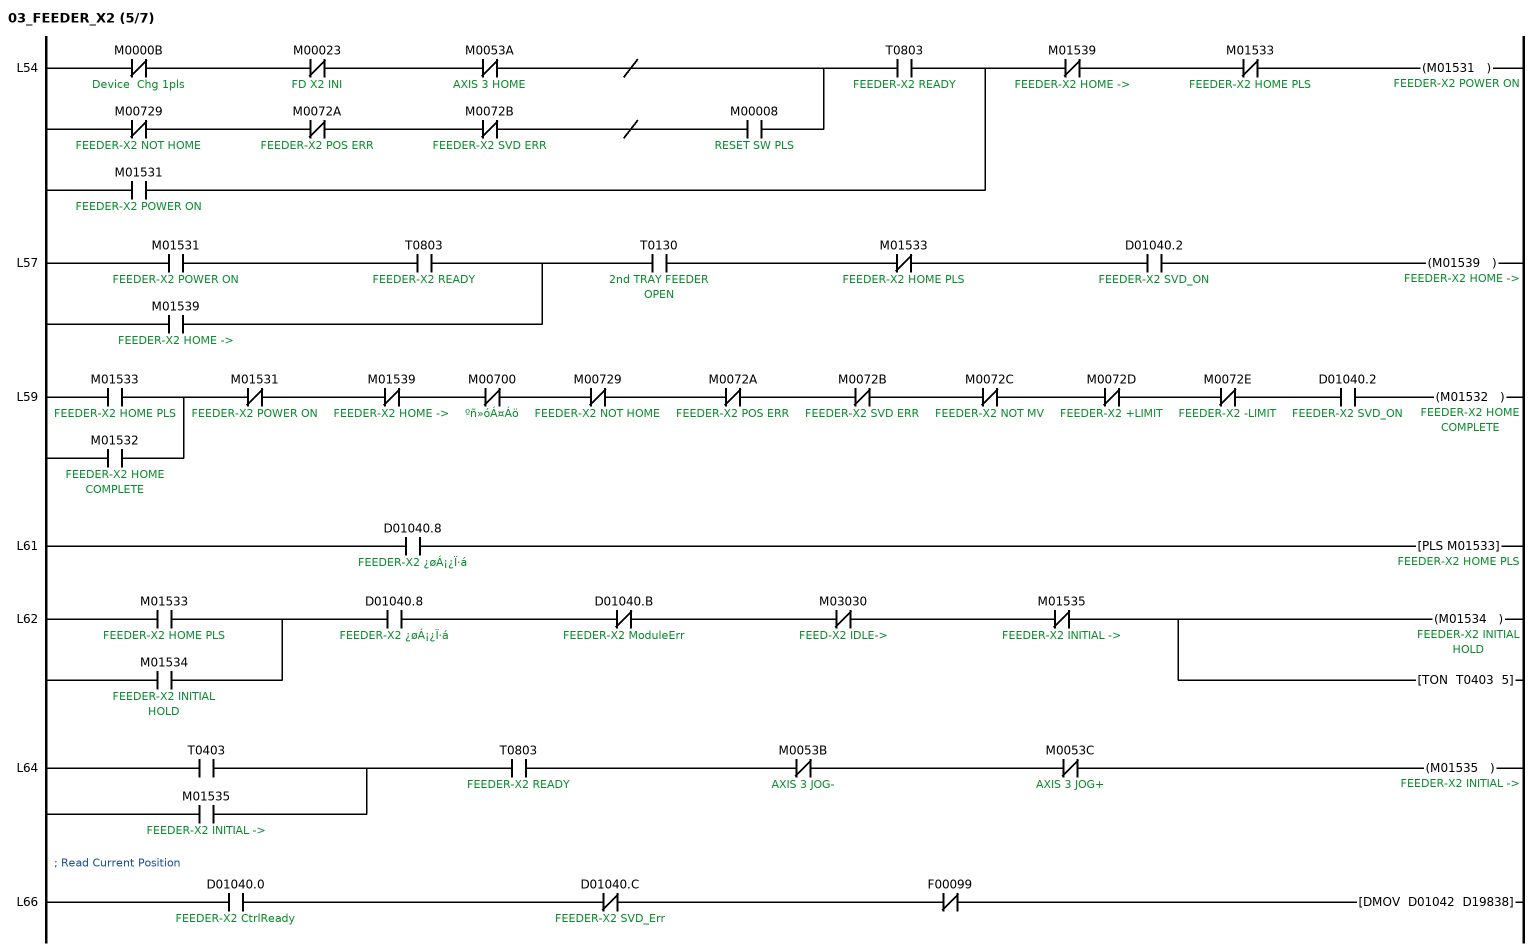
[picture p24: 03_FEEDER_X2 rungs L54-L66]
; L54
LOAD NOT  M0000B	// Device  Chg 1pls
AND NOT   M00023	// FD X2 INI
AND NOT   M0053A	// AXIS 3 HOME
NOT
LOAD NOT  M00729	// FEEDER-X2 NOT HOME
AND NOT   M0072A	// FEEDER-X2 POS ERR
AND NOT   M0072B	// FEEDER-X2 SVD ERR
NOT
AND       M00008	// RESET SW PLS
OR LOAD
AND       T0803	// FEEDER-X2 READY
OR        M01531	// FEEDER-X2 POWER ON
AND NOT   M01539	// FEEDER-X2 HOME ->
AND NOT   M01533	// FEEDER-X2 HOME PLS
OUT       M01531	// FEEDER-X2 POWER ON
; L57
LOAD      M01531	// FEEDER-X2 POWER ON
AND       T0803	// FEEDER-X2 READY
OR        M01539	// FEEDER-X2 HOME ->
AND       T0130	// 2nd TRAY FEEDER OPEN
AND NOT   M01533	// FEEDER-X2 HOME PLS
AND       D01040.2	// FEEDER-X2 SVD_ON
OUT       M01539	// FEEDER-X2 HOME ->
; L59
LOAD      M01533	// FEEDER-X2 HOME PLS
OR        M01532	// FEEDER-X2 HOME COMPLETE
AND NOT   M01531	// FEEDER-X2 POWER ON
AND NOT   M01539	// FEEDER-X2 HOME ->
AND NOT   M00700	// ºñ»óÁ¤Áö
AND NOT   M00729	// FEEDER-X2 NOT HOME
AND NOT   M0072A	// FEEDER-X2 POS ERR
AND NOT   M0072B	// FEEDER-X2 SVD ERR
AND NOT   M0072C	// FEEDER-X2 NOT MV
AND NOT   M0072D	// FEEDER-X2 +LIMIT
AND NOT   M0072E	// FEEDER-X2 -LIMIT
AND       D01040.2	// FEEDER-X2 SVD_ON
OUT       M01532	// FEEDER-X2 HOME COMPLETE
; L61
LOAD      D01040.8	// FEEDER-X2 ¿øÁ¡¿Ï·á
OUTP      M01533	// FEEDER-X2 HOME PLS
; L62
LOAD      M01533	// FEEDER-X2 HOME PLS
OR        M01534	// FEEDER-X2 INITIAL HOLD
AND       D01040.8	// FEEDER-X2 ¿øÁ¡¿Ï·á
AND NOT   D01040.B	// FEEDER-X2 ModuleErr
AND NOT   M03030	// FEED-X2 IDLE->
AND NOT   M01535	// FEEDER-X2 INITIAL ->
OUT       M01534	// FEEDER-X2 INITIAL HOLD
TON       T0403 5
; L64
LOAD      T0403
OR        M01535	// FEEDER-X2 INITIAL ->
AND       T0803	// FEEDER-X2 READY
AND NOT   M0053B	// AXIS 3 JOG-
AND NOT   M0053C	// AXIS 3 JOG+
OUT       M01535	// FEEDER-X2 INITIAL ->
; L66
LOAD      D01040.0	// FEEDER-X2 CtrlReady
AND NOT   D01040.C	// FEEDER-X2 SVD_Err
AND NOT   F00099
DMOV      D01042 D19838
// output comment: Read Current Position

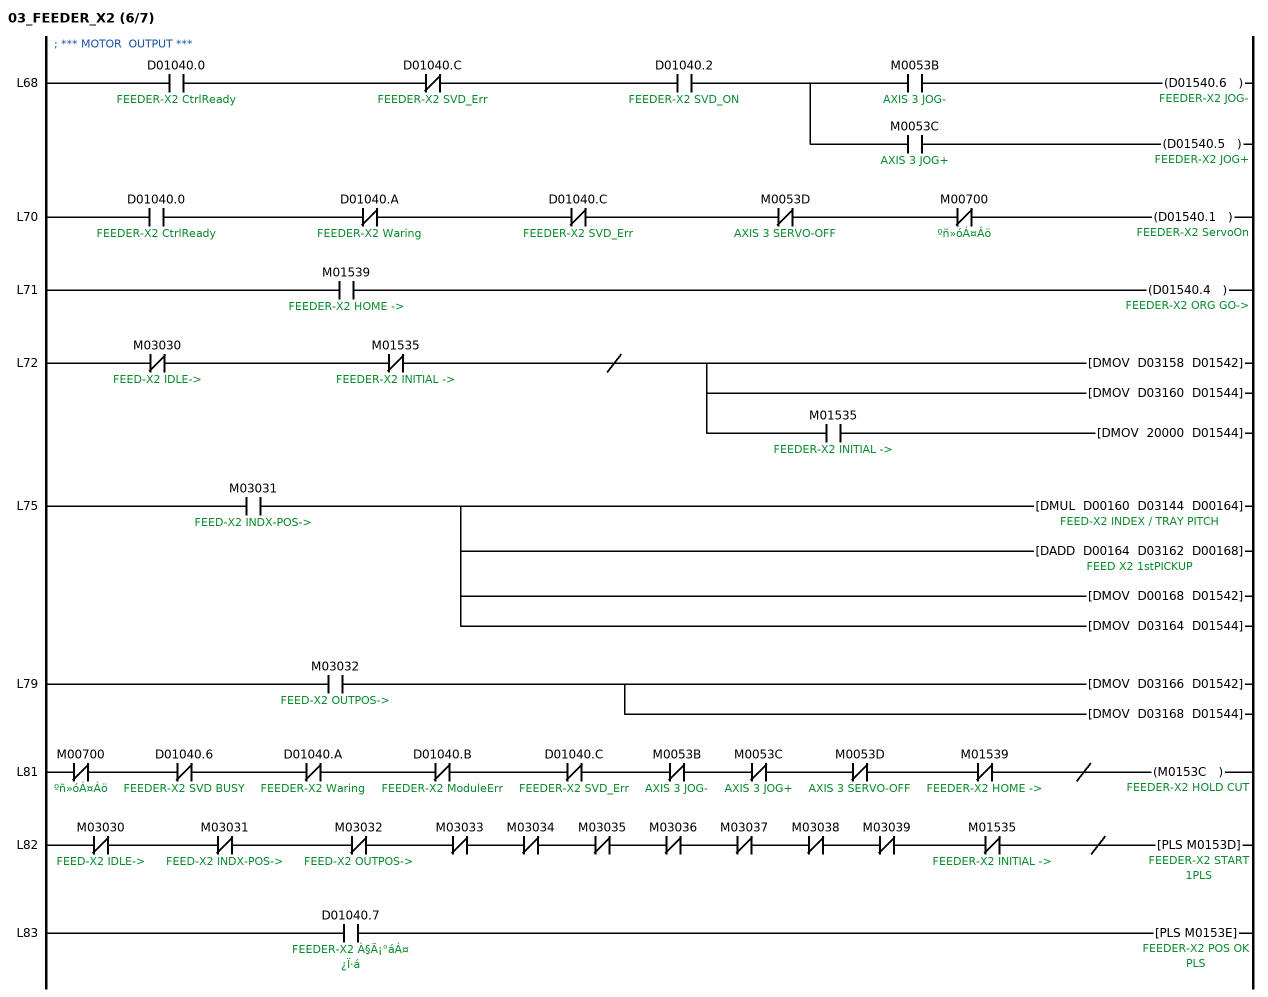
// *** MOTOR  OUTPUT ***
; L68
LOAD      D01040.0	// FEEDER-X2 CtrlReady
AND NOT   D01040.C	// FEEDER-X2 SVD_Err
AND       D01040.2	// FEEDER-X2 SVD_ON
MPUSH
AND       M0053B	// AXIS 3 JOG-
OUT       D01540.6	// FEEDER-X2 JOG-
MPOP
AND       M0053C	// AXIS 3 JOG+
OUT       D01540.5	// FEEDER-X2 JOG+
; L70
LOAD      D01040.0	// FEEDER-X2 CtrlReady
AND NOT   D01040.A	// FEEDER-X2 Waring
AND NOT   D01040.C	// FEEDER-X2 SVD_Err
AND NOT   M0053D	// AXIS 3 SERVO-OFF
AND NOT   M00700	// ºñ»óÁ¤Áö
OUT       D01540.1	// FEEDER-X2 ServoOn
; L71
LOAD      M01539	// FEEDER-X2 HOME ->
OUT       D01540.4	// FEEDER-X2 ORG GO->
; L72
LOAD NOT  M03030	// FEED-X2 IDLE->
AND NOT   M01535	// FEEDER-X2 INITIAL ->
NOT
DMOV      D03158 D01542
DMOV      D03160 D01544
AND       M01535	// FEEDER-X2 INITIAL ->
DMOV      20000 D01544
; L75
LOAD      M03031	// FEED-X2 INDX-POS->
DMUL      D00160 D03144 D00164	// FEED-X2 INDEX / TRAY PITCH
DADD      D00164 D03162 D00168	// FEED X2 1stPICKUP
DMOV      D00168 D01542
DMOV      D03164 D01544
; L79
LOAD      M03032	// FEED-X2 OUTPOS->
DMOV      D03166 D01542
DMOV      D03168 D01544
; L81
LOAD NOT  M00700	// ºñ»óÁ¤Áö
AND NOT   D01040.6	// FEEDER-X2 SVD BUSY
AND NOT   D01040.A	// FEEDER-X2 Waring
AND NOT   D01040.B	// FEEDER-X2 ModuleErr
AND NOT   D01040.C	// FEEDER-X2 SVD_Err
AND NOT   M0053B	// AXIS 3 JOG-
AND NOT   M0053C	// AXIS 3 JOG+
AND NOT   M0053D	// AXIS 3 SERVO-OFF
AND NOT   M01539	// FEEDER-X2 HOME ->
NOT
OUT       M0153C	// FEEDER-X2 HOLD CUT
; L82
LOAD NOT  M03030	// FEED-X2 IDLE->
AND NOT   M03031	// FEED-X2 INDX-POS->
AND NOT   M03032	// FEED-X2 OUTPOS->
AND NOT   M03033
AND NOT   M03034
AND NOT   M03035
AND NOT   M03036
AND NOT   M03037
AND NOT   M03038
AND NOT   M03039
AND NOT   M01535	// FEEDER-X2 INITIAL ->
NOT
OUTP      M0153D	// FEEDER-X2 START 1PLS
; L83
LOAD      D01040.7	// FEEDER-X2 À§Ä¡°áÁ¤ ¿Ï·á
OUTP      M0153E	// FEEDER-X2 POS OK PLS

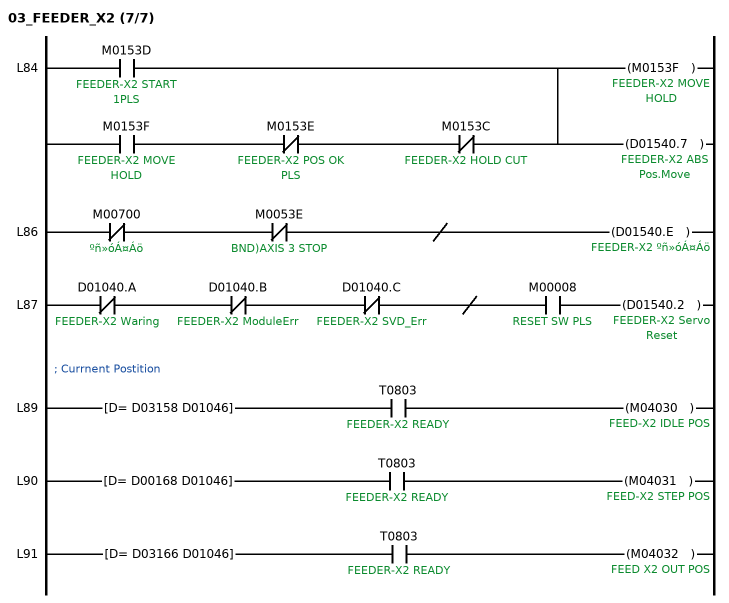
; L84
LOAD      M0153D	// FEEDER-X2 START 1PLS
LOAD      M0153F	// FEEDER-X2 MOVE HOLD
AND NOT   M0153E	// FEEDER-X2 POS OK PLS
AND NOT   M0153C	// FEEDER-X2 HOLD CUT
OR LOAD
OUT       M0153F	// FEEDER-X2 MOVE HOLD
OUT       D01540.7	// FEEDER-X2 ABS Pos.Move
; L86
LOAD NOT  M00700	// ºñ»óÁ¤Áö
AND NOT   M0053E	// BND)AXIS 3 STOP
NOT
OUT       D01540.E	// FEEDER-X2 ºñ»óÁ¤Áö
; L87
LOAD NOT  D01040.A	// FEEDER-X2 Waring
AND NOT   D01040.B	// FEEDER-X2 ModuleErr
AND NOT   D01040.C	// FEEDER-X2 SVD_Err
NOT
AND       M00008	// RESET SW PLS
OUT       D01540.2	// FEEDER-X2 Servo Reset
// Currnent Postition
; L89
LOADD=    D03158 D01046
AND       T0803	// FEEDER-X2 READY
OUT       M04030	// FEED-X2 IDLE POS
; L90
LOADD=    D00168 D01046
AND       T0803	// FEEDER-X2 READY
OUT       M04031	// FEED-X2 STEP POS
; L91
LOADD=    D03166 D01046
AND       T0803	// FEEDER-X2 READY
OUT       M04032	// FEED X2 OUT POS

PROGRAM 04_PICKER_Y (task: ½ºÄµ ÇÁ·Î±×·¥)

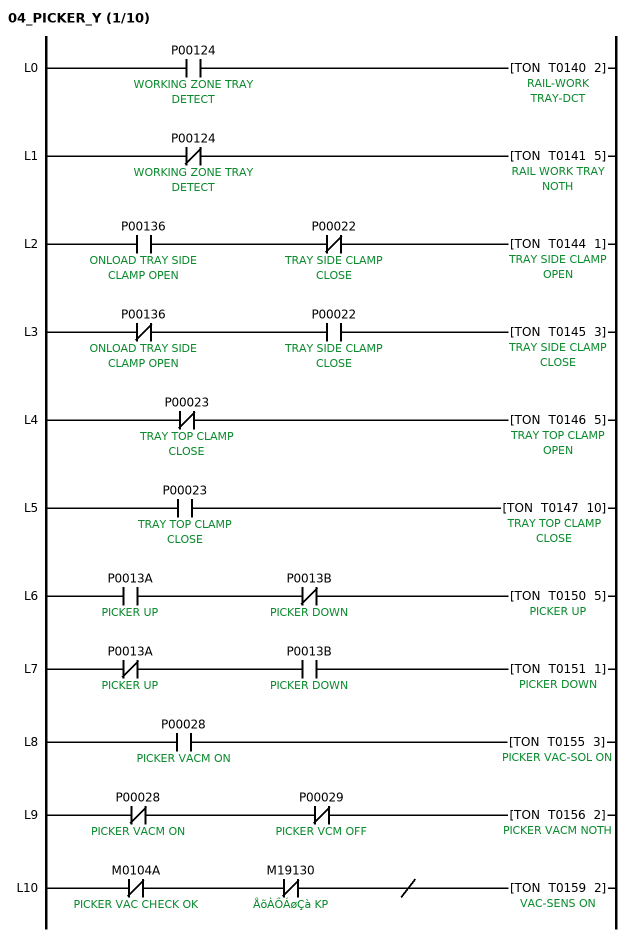
; L0
LOAD      P00124	// WORKING ZONE TRAY DETECT
TON       T0140 2	// RAIL-WORK TRAY-DCT
; L1
LOAD NOT  P00124	// WORKING ZONE TRAY DETECT
TON       T0141 5	// RAIL WORK TRAY NOTH
; L2
LOAD      P00136	// ONLOAD TRAY SIDE CLAMP OPEN
AND NOT   P00022	// TRAY SIDE CLAMP CLOSE
TON       T0144 1	// TRAY SIDE CLAMP OPEN
; L3
LOAD NOT  P00136	// ONLOAD TRAY SIDE CLAMP OPEN
AND       P00022	// TRAY SIDE CLAMP CLOSE
TON       T0145 3	// TRAY SIDE CLAMP CLOSE
; L4
LOAD NOT  P00023	// TRAY TOP CLAMP CLOSE
TON       T0146 5	// TRAY TOP CLAMP OPEN
; L5
LOAD      P00023	// TRAY TOP CLAMP CLOSE
TON       T0147 10	// TRAY TOP CLAMP CLOSE
; L6
LOAD      P0013A	// PICKER UP
AND NOT   P0013B	// PICKER DOWN
TON       T0150 5	// PICKER UP
; L7
LOAD NOT  P0013A	// PICKER UP
AND       P0013B	// PICKER DOWN
TON       T0151 1	// PICKER DOWN
; L8
LOAD      P00028	// PICKER VACM ON
TON       T0155 3	// PICKER VAC-SOL ON
; L9
LOAD NOT  P00028	// PICKER VACM ON
AND NOT   P00029	// PICKER VCM OFF
TON       T0156 2	// PICKER VACM NOTH
; L10
LOAD NOT  M0104A	// PICKER VAC CHECK OK
AND NOT   M19130	// ÅõÀÔÁøÇà KP
NOT
TON       T0159 2	// VAC-SENS ON

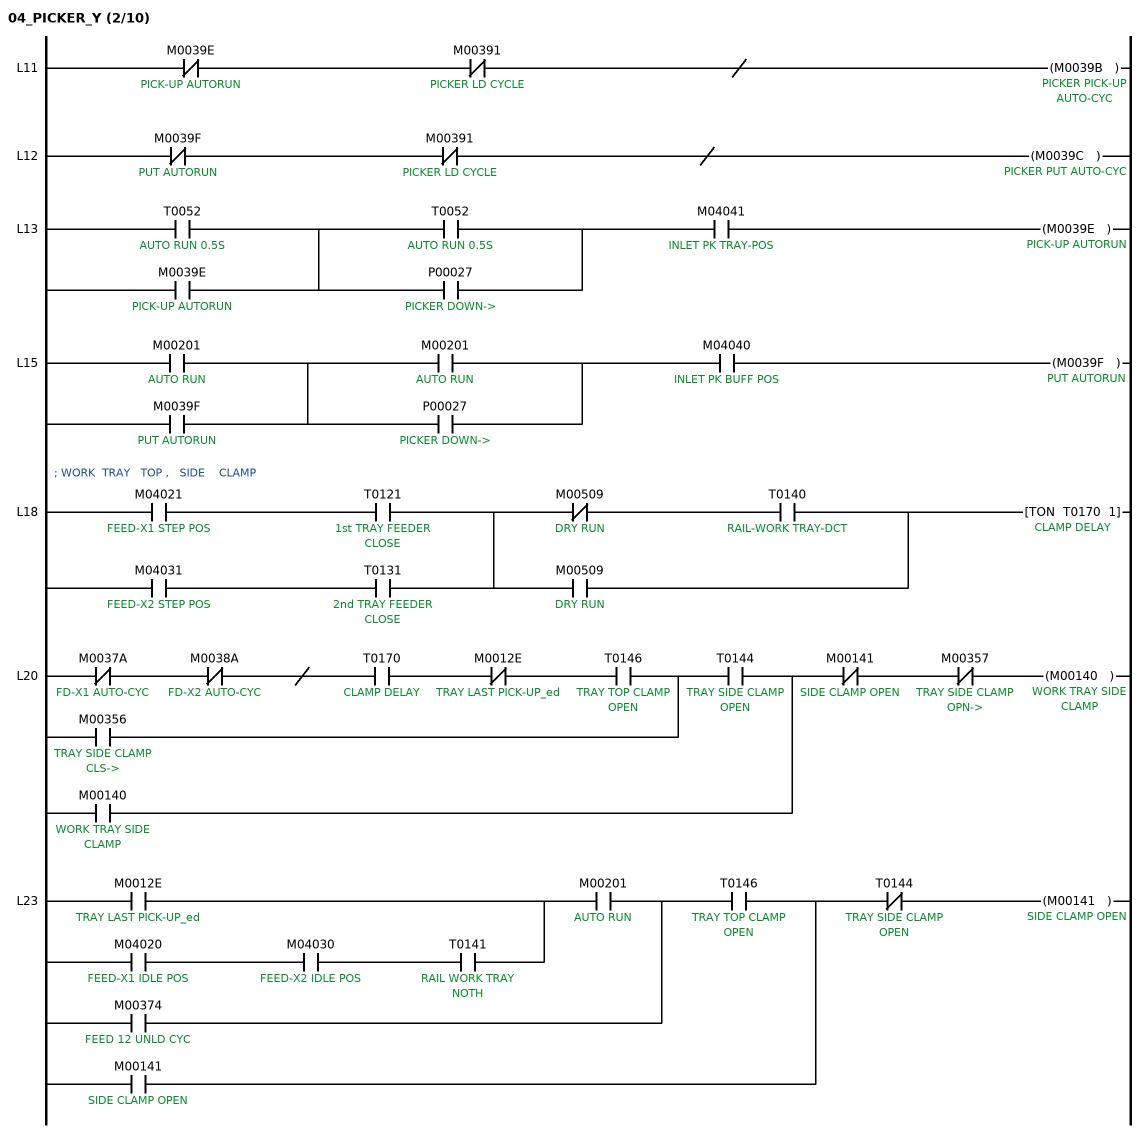
; L11
LOAD NOT  M0039E	// PICK-UP AUTORUN
AND NOT   M00391	// PICKER LD CYCLE
NOT
OUT       M0039B	// PICKER PICK-UP AUTO-CYC
; L12
LOAD NOT  M0039F	// PUT AUTORUN
AND NOT   M00391	// PICKER LD CYCLE
NOT
OUT       M0039C	// PICKER PUT AUTO-CYC
; L13
LOAD      T0052	// AUTO RUN 0.5S
OR        M0039E	// PICK-UP AUTORUN
LOAD      T0052	// AUTO RUN 0.5S
OR        P00027	// PICKER DOWN->
AND LOAD
AND       M04041	// INLET PK TRAY-POS
OUT       M0039E	// PICK-UP AUTORUN
; L15
LOAD      M00201	// AUTO RUN
OR        M0039F	// PUT AUTORUN
LOAD      M00201	// AUTO RUN
OR        P00027	// PICKER DOWN->
AND LOAD
AND       M04040	// INLET PK BUFF POS
OUT       M0039F	// PUT AUTORUN
// WORK  TRAY   TOP ,   SIDE    CLAMP
; L18
LOAD      M04021	// FEED-X1 STEP POS
AND       T0121	// 1st TRAY FEEDER CLOSE
LOAD      M04031	// FEED-X2 STEP POS
AND       T0131	// 2nd TRAY FEEDER CLOSE
OR LOAD
LOAD NOT  M00509	// DRY RUN
AND       T0140	// RAIL-WORK TRAY-DCT
OR        M00509	// DRY RUN
AND LOAD
TON       T0170 1	// CLAMP DELAY
; L20
LOAD NOT  M0037A	// FD-X1 AUTO-CYC
AND NOT   M0038A	// FD-X2 AUTO-CYC
NOT
AND       T0170	// CLAMP DELAY
AND NOT   M0012E	// TRAY LAST PICK-UP_ed
AND       T0146	// TRAY TOP CLAMP OPEN
OR        M00356	// TRAY SIDE CLAMP CLS->
AND       T0144	// TRAY SIDE CLAMP OPEN
OR        M00140	// WORK TRAY SIDE CLAMP
AND NOT   M00141	// SIDE CLAMP OPEN
AND NOT   M00357	// TRAY SIDE CLAMP OPN->
OUT       M00140	// WORK TRAY SIDE CLAMP
; L23
LOAD      M0012E	// TRAY LAST PICK-UP_ed
LOAD      M04020	// FEED-X1 IDLE POS
AND       M04030	// FEED-X2 IDLE POS
AND       T0141	// RAIL WORK TRAY NOTH
OR LOAD
AND       M00201	// AUTO RUN
OR        M00374	// FEED 12 UNLD CYC
AND       T0146	// TRAY TOP CLAMP OPEN
OR        M00141	// SIDE CLAMP OPEN
AND NOT   T0144	// TRAY SIDE CLAMP OPEN
OUT       M00141	// SIDE CLAMP OPEN

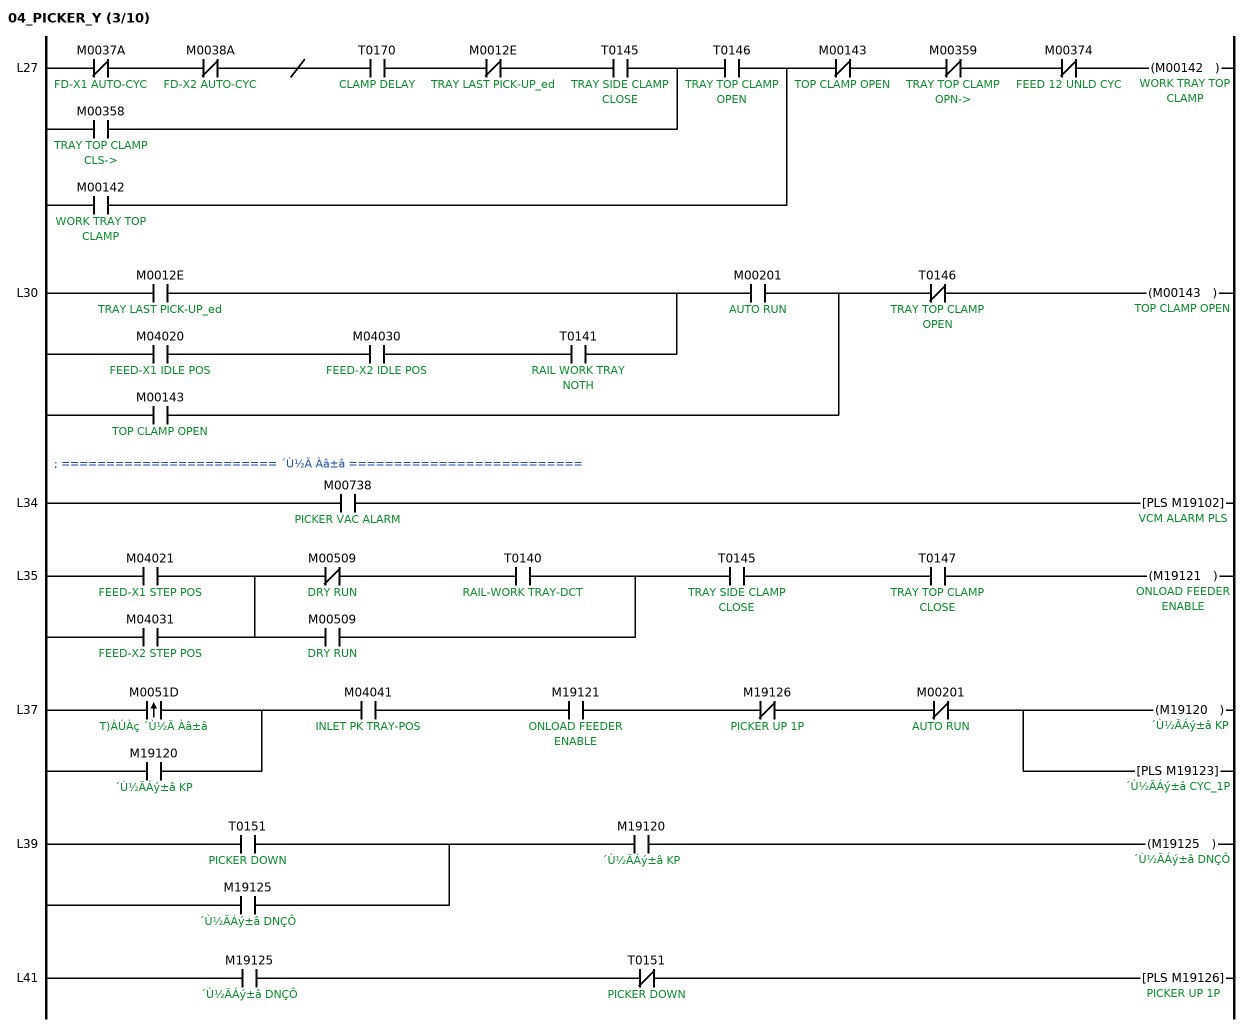
; L27
LOAD NOT  M0037A	// FD-X1 AUTO-CYC
AND NOT   M0038A	// FD-X2 AUTO-CYC
NOT
AND       T0170	// CLAMP DELAY
AND NOT   M0012E	// TRAY LAST PICK-UP_ed
AND       T0145	// TRAY SIDE CLAMP CLOSE
OR        M00358	// TRAY TOP CLAMP CLS->
AND       T0146	// TRAY TOP CLAMP OPEN
OR        M00142	// WORK TRAY TOP CLAMP
AND NOT   M00143	// TOP CLAMP OPEN
AND NOT   M00359	// TRAY TOP CLAMP OPN->
AND NOT   M00374	// FEED 12 UNLD CYC
OUT       M00142	// WORK TRAY TOP CLAMP
; L30
LOAD      M0012E	// TRAY LAST PICK-UP_ed
LOAD      M04020	// FEED-X1 IDLE POS
AND       M04030	// FEED-X2 IDLE POS
AND       T0141	// RAIL WORK TRAY NOTH
OR LOAD
AND       M00201	// AUTO RUN
OR        M00143	// TOP CLAMP OPEN
AND NOT   T0146	// TRAY TOP CLAMP OPEN
OUT       M00143	// TOP CLAMP OPEN
// ======================== ´Ù½Ã Àâ±â ==========================
; L34
LOAD      M00738	// PICKER VAC ALARM
OUTP      M19102	// VCM ALARM PLS
; L35
LOAD      M04021	// FEED-X1 STEP POS
OR        M04031	// FEED-X2 STEP POS
LOAD NOT  M00509	// DRY RUN
AND       T0140	// RAIL-WORK TRAY-DCT
OR        M00509	// DRY RUN
AND LOAD
AND       T0145	// TRAY SIDE CLAMP CLOSE
AND       T0147	// TRAY TOP CLAMP CLOSE
OUT       M19121	// ONLOAD FEEDER ENABLE
; L37
LOADP     M0051D	// T)ÀÚÀç ´Ù½Ã Àâ±â
OR        M19120	// ´Ù½ÃÁý±â KP
AND       M04041	// INLET PK TRAY-POS
AND       M19121	// ONLOAD FEEDER ENABLE
AND NOT   M19126	// PICKER UP 1P
AND NOT   M00201	// AUTO RUN
OUT       M19120	// ´Ù½ÃÁý±â KP
OUTP      M19123	// ´Ù½ÃÁý±â CYC_1P
; L39
LOAD      T0151	// PICKER DOWN
OR        M19125	// ´Ù½ÃÁý±â DNÇÔ
AND       M19120	// ´Ù½ÃÁý±â KP
OUT       M19125	// ´Ù½ÃÁý±â DNÇÔ
; L41
LOAD      M19125	// ´Ù½ÃÁý±â DNÇÔ
AND NOT   T0151	// PICKER DOWN
OUTP      M19126	// PICKER UP 1P

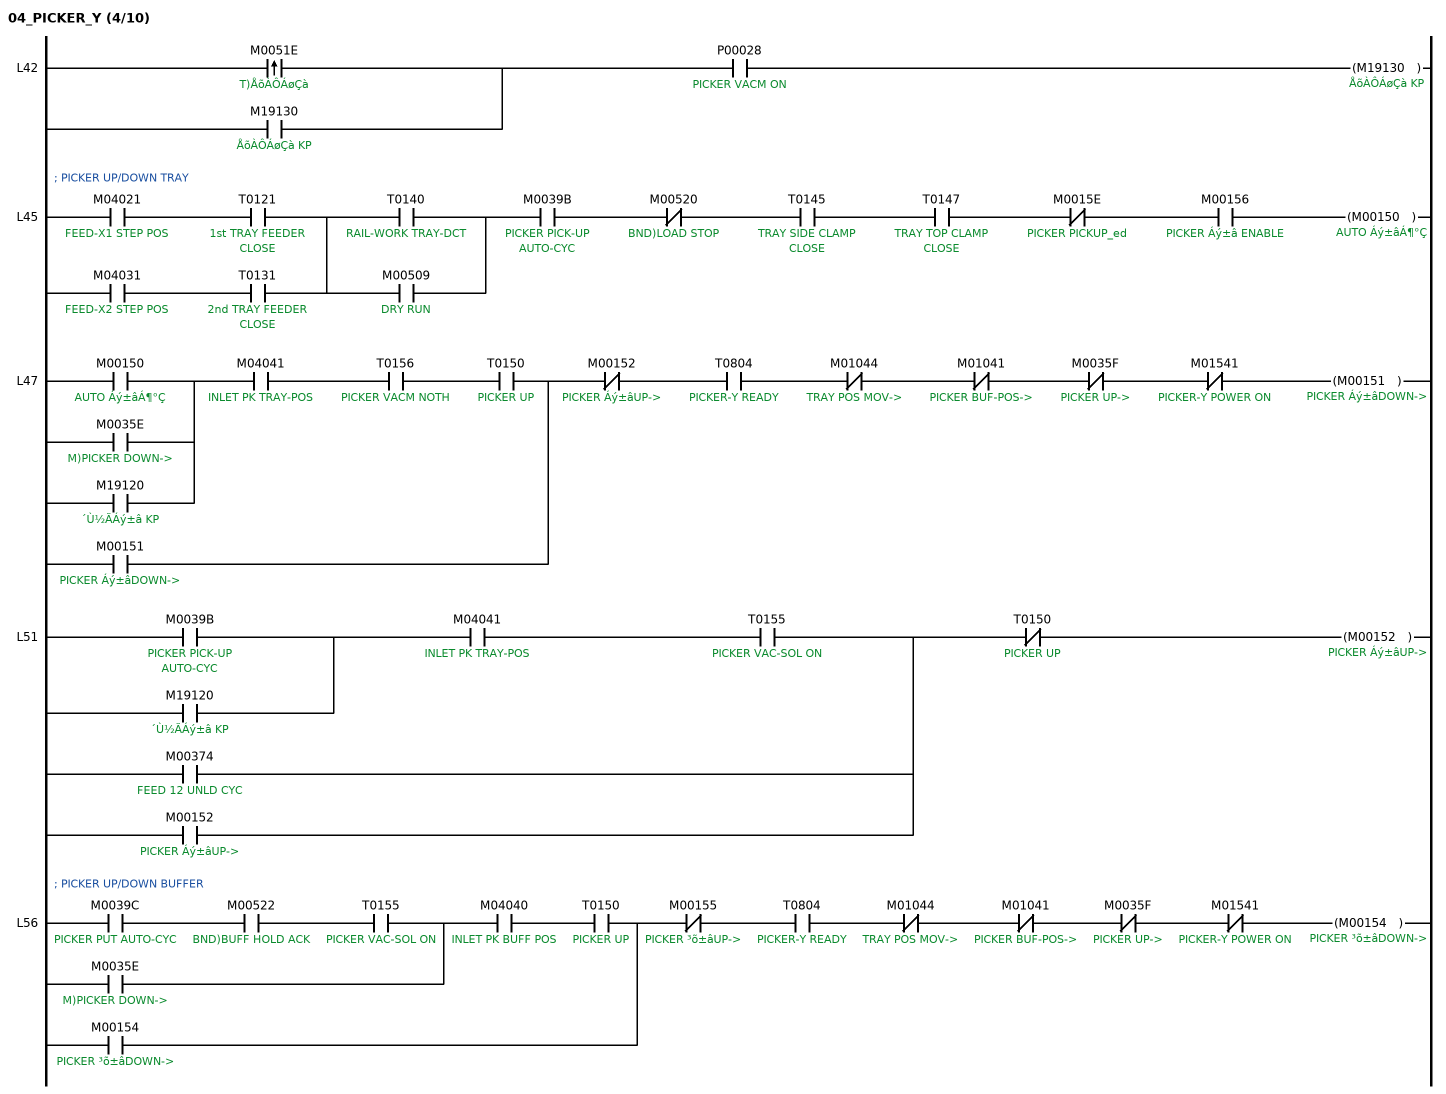
; L42
LOADP     M0051E	// T)ÅõÀÔÁøÇà
OR        M19130	// ÅõÀÔÁøÇà KP
AND       P00028	// PICKER VACM ON
OUT       M19130	// ÅõÀÔÁøÇà KP
// PICKER UP/DOWN TRAY
; L45
LOAD      M04021	// FEED-X1 STEP POS
AND       T0121	// 1st TRAY FEEDER CLOSE
LOAD      M04031	// FEED-X2 STEP POS
AND       T0131	// 2nd TRAY FEEDER CLOSE
OR LOAD
LOAD      T0140	// RAIL-WORK TRAY-DCT
OR        M00509	// DRY RUN
AND LOAD
AND       M0039B	// PICKER PICK-UP AUTO-CYC
AND NOT   M00520	// BND)LOAD STOP
AND       T0145	// TRAY SIDE CLAMP CLOSE
AND       T0147	// TRAY TOP CLAMP CLOSE
AND NOT   M0015E	// PICKER PICKUP_ed
AND       M00156	// PICKER Áý±â ENABLE
OUT       M00150	// AUTO Áý±âÁ¶°Ç
; L47
LOAD      M00150	// AUTO Áý±âÁ¶°Ç
OR        M0035E	// M)PICKER DOWN->
OR        M19120	// ´Ù½ÃÁý±â KP
AND       M04041	// INLET PK TRAY-POS
AND       T0156	// PICKER VACM NOTH
AND       T0150	// PICKER UP
OR        M00151	// PICKER Áý±âDOWN->
AND NOT   M00152	// PICKER Áý±âUP->
AND       T0804	// PICKER-Y READY
AND NOT   M01044	// TRAY POS MOV->
AND NOT   M01041	// PICKER BUF-POS->
AND NOT   M0035F	// PICKER UP->
AND NOT   M01541	// PICKER-Y POWER ON
OUT       M00151	// PICKER Áý±âDOWN->
; L51
LOAD      M0039B	// PICKER PICK-UP AUTO-CYC
OR        M19120	// ´Ù½ÃÁý±â KP
AND       M04041	// INLET PK TRAY-POS
AND       T0155	// PICKER VAC-SOL ON
OR        M00374	// FEED 12 UNLD CYC
OR        M00152	// PICKER Áý±âUP->
AND NOT   T0150	// PICKER UP
OUT       M00152	// PICKER Áý±âUP->
// PICKER UP/DOWN BUFFER
; L56
LOAD      M0039C	// PICKER PUT AUTO-CYC
AND       M00522	// BND)BUFF HOLD ACK
AND       T0155	// PICKER VAC-SOL ON
OR        M0035E	// M)PICKER DOWN->
AND       M04040	// INLET PK BUFF POS
AND       T0150	// PICKER UP
OR        M00154	// PICKER ³õ±âDOWN->
AND NOT   M00155	// PICKER ³õ±âUP->
AND       T0804	// PICKER-Y READY
AND NOT   M01044	// TRAY POS MOV->
AND NOT   M01041	// PICKER BUF-POS->
AND NOT   M0035F	// PICKER UP->
AND NOT   M01541	// PICKER-Y POWER ON
OUT       M00154	// PICKER ³õ±âDOWN->

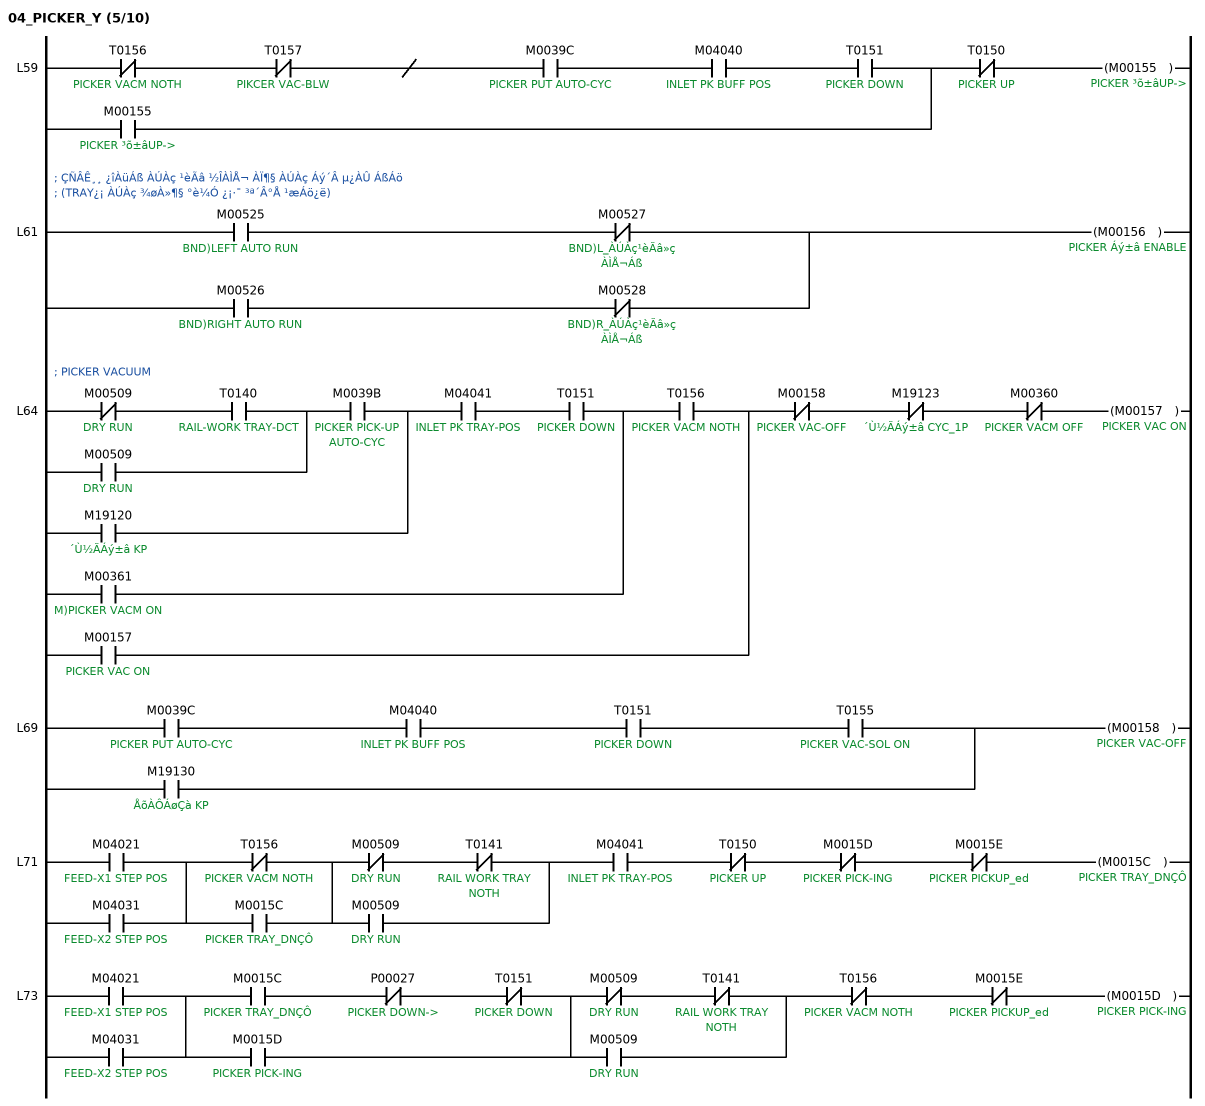
; L59
LOAD NOT  T0156	// PICKER VACM NOTH
AND NOT   T0157	// PIKCER VAC-BLW
NOT
AND       M0039C	// PICKER PUT AUTO-CYC
AND       M04040	// INLET PK BUFF POS
AND       T0151	// PICKER DOWN
OR        M00155	// PICKER ³õ±âUP->
AND NOT   T0150	// PICKER UP
OUT       M00155	// PICKER ³õ±âUP->
; L61
LOAD      M00525	// BND)LEFT AUTO RUN
AND NOT   M00527	// BND)L_ÀÚÀç¹èÃâ»çÀÌÅ¬Áß
LOAD      M00526	// BND)RIGHT AUTO RUN
AND NOT   M00528	// BND)R_ÀÚÀç¹èÃâ»çÀÌÅ¬Áß
OR LOAD
OUT       M00156	// PICKER Áý±â ENABLE
// output comment: ÇÑÂÊ¸¸ ¿îÀüÁß ÀÚÀç ¹èÃâ ½ÎÀÌÅ¬ ÀÏ¶§ ÀÚÀç Áý´Â µ¿ÀÛ ÁßÁö (TRAY¿¡ ÀÚÀç ¾øÀ»¶§ °è¼Ó ¿¡·¯ ³ª´Â°Å ¹æÁö¿ë)
// PICKER VACUUM
; L64
LOAD NOT  M00509	// DRY RUN
AND       T0140	// RAIL-WORK TRAY-DCT
OR        M00509	// DRY RUN
AND       M0039B	// PICKER PICK-UP AUTO-CYC
OR        M19120	// ´Ù½ÃÁý±â KP
AND       M04041	// INLET PK TRAY-POS
AND       T0151	// PICKER DOWN
OR        M00361	// M)PICKER VACM ON
AND       T0156	// PICKER VACM NOTH
OR        M00157	// PICKER VAC ON
AND NOT   M00158	// PICKER VAC-OFF
AND NOT   M19123	// ´Ù½ÃÁý±â CYC_1P
AND NOT   M00360	// PICKER VACM OFF
OUT       M00157	// PICKER VAC ON
; L69
LOAD      M0039C	// PICKER PUT AUTO-CYC
AND       M04040	// INLET PK BUFF POS
AND       T0151	// PICKER DOWN
AND       T0155	// PICKER VAC-SOL ON
OR        M19130	// ÅõÀÔÁøÇà KP
OUT       M00158	// PICKER VAC-OFF
; L71
LOAD      M04021	// FEED-X1 STEP POS
OR        M04031	// FEED-X2 STEP POS
LOAD NOT  T0156	// PICKER VACM NOTH
OR        M0015C	// PICKER TRAY_DNÇÔ
AND LOAD
LOAD NOT  M00509	// DRY RUN
AND NOT   T0141	// RAIL WORK TRAY NOTH
OR        M00509	// DRY RUN
AND LOAD
AND       M04041	// INLET PK TRAY-POS
AND NOT   T0150	// PICKER UP
AND NOT   M0015D	// PICKER PICK-ING
AND NOT   M0015E	// PICKER PICKUP_ed
OUT       M0015C	// PICKER TRAY_DNÇÔ
; L73
LOAD      M04021	// FEED-X1 STEP POS
OR        M04031	// FEED-X2 STEP POS
LOAD      M0015C	// PICKER TRAY_DNÇÔ
AND NOT   P00027	// PICKER DOWN->
AND NOT   T0151	// PICKER DOWN
OR        M0015D	// PICKER PICK-ING
AND LOAD
LOAD NOT  M00509	// DRY RUN
AND NOT   T0141	// RAIL WORK TRAY NOTH
OR        M00509	// DRY RUN
AND LOAD
AND NOT   T0156	// PICKER VACM NOTH
AND NOT   M0015E	// PICKER PICKUP_ed
OUT       M0015D	// PICKER PICK-ING

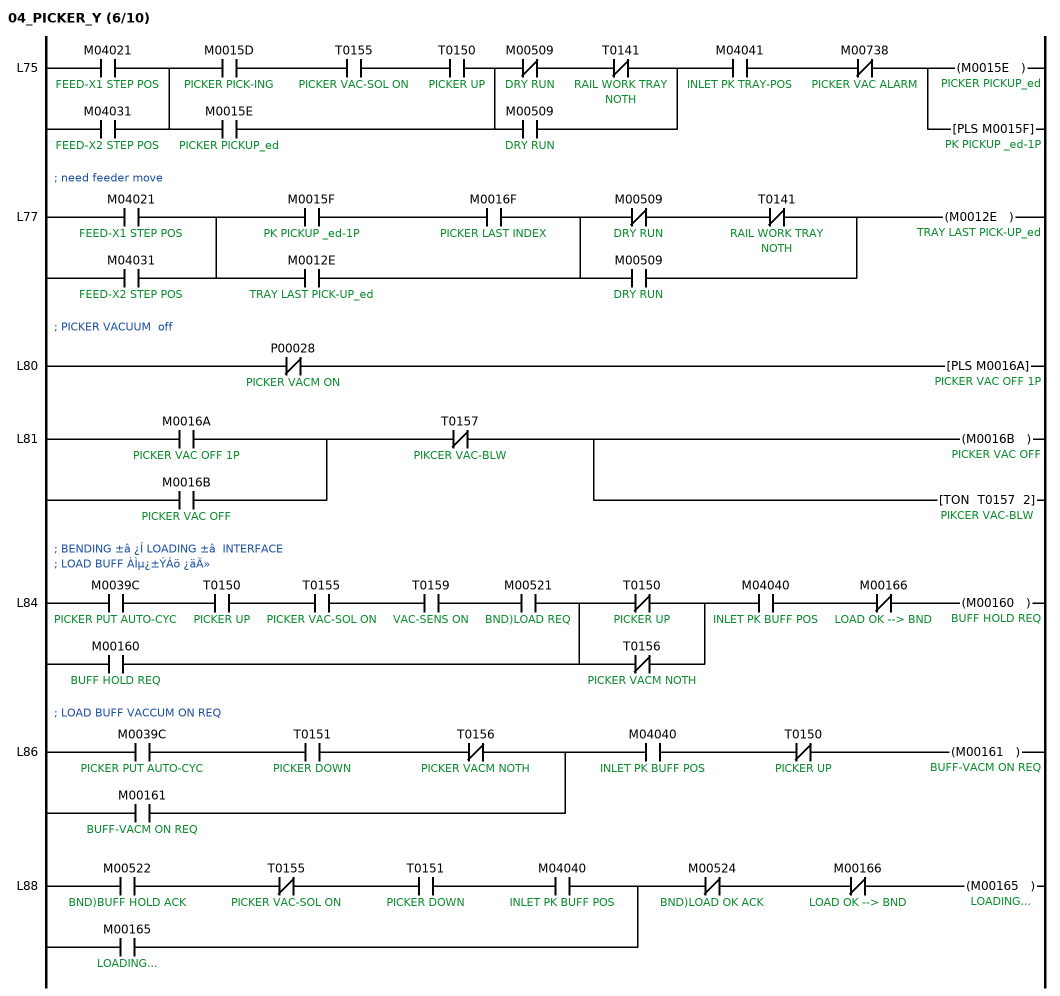
; L75
LOAD      M04021	// FEED-X1 STEP POS
OR        M04031	// FEED-X2 STEP POS
LOAD      M0015D	// PICKER PICK-ING
AND       T0155	// PICKER VAC-SOL ON
AND       T0150	// PICKER UP
OR        M0015E	// PICKER PICKUP_ed
AND LOAD
LOAD NOT  M00509	// DRY RUN
AND NOT   T0141	// RAIL WORK TRAY NOTH
OR        M00509	// DRY RUN
AND LOAD
AND       M04041	// INLET PK TRAY-POS
AND NOT   M00738	// PICKER VAC ALARM
OUT       M0015E	// PICKER PICKUP_ed
OUTP      M0015F	// PK PICKUP _ed-1P
; L77
LOAD      M04021	// FEED-X1 STEP POS
OR        M04031	// FEED-X2 STEP POS
LOAD      M0015F	// PK PICKUP _ed-1P
AND       M0016F	// PICKER LAST INDEX
OR        M0012E	// TRAY LAST PICK-UP_ed
AND LOAD
LOAD NOT  M00509	// DRY RUN
AND NOT   T0141	// RAIL WORK TRAY NOTH
OR        M00509	// DRY RUN
AND LOAD
OUT       M0012E	// TRAY LAST PICK-UP_ed
// output comment: need feeder move
// PICKER VACUUM  off
; L80
LOAD NOT  P00028	// PICKER VACM ON
OUTP      M0016A	// PICKER VAC OFF 1P
; L81
LOAD      M0016A	// PICKER VAC OFF 1P
OR        M0016B	// PICKER VAC OFF
AND NOT   T0157	// PIKCER VAC-BLW
OUT       M0016B	// PICKER VAC OFF
TON       T0157 2	// PIKCER VAC-BLW
// BENDING ±â ¿Í LOADING ±â  INTERFACE
; L84
LOAD      M0039C	// PICKER PUT AUTO-CYC
AND       T0150	// PICKER UP
AND       T0155	// PICKER VAC-SOL ON
AND       T0159	// VAC-SENS ON
AND       M00521	// BND)LOAD REQ
OR        M00160	// BUFF HOLD REQ
LOAD NOT  T0150	// PICKER UP
OR NOT    T0156	// PICKER VACM NOTH
AND LOAD
AND       M04040	// INLET PK BUFF POS
AND NOT   M00166	// LOAD OK --> BND
OUT       M00160	// BUFF HOLD REQ
// output comment: LOAD BUFF ÀÌµ¿±ÝÁö ¿äÃ»
; L86
LOAD      M0039C	// PICKER PUT AUTO-CYC
AND       T0151	// PICKER DOWN
AND NOT   T0156	// PICKER VACM NOTH
OR        M00161	// BUFF-VACM ON REQ
AND       M04040	// INLET PK BUFF POS
AND NOT   T0150	// PICKER UP
OUT       M00161	// BUFF-VACM ON REQ
// output comment: LOAD BUFF VACCUM ON REQ
; L88
LOAD      M00522	// BND)BUFF HOLD ACK
AND NOT   T0155	// PICKER VAC-SOL ON
AND       T0151	// PICKER DOWN
AND       M04040	// INLET PK BUFF POS
OR        M00165	// LOADING...
AND NOT   M00524	// BND)LOAD OK ACK
AND NOT   M00166	// LOAD OK --> BND
OUT       M00165	// LOADING...

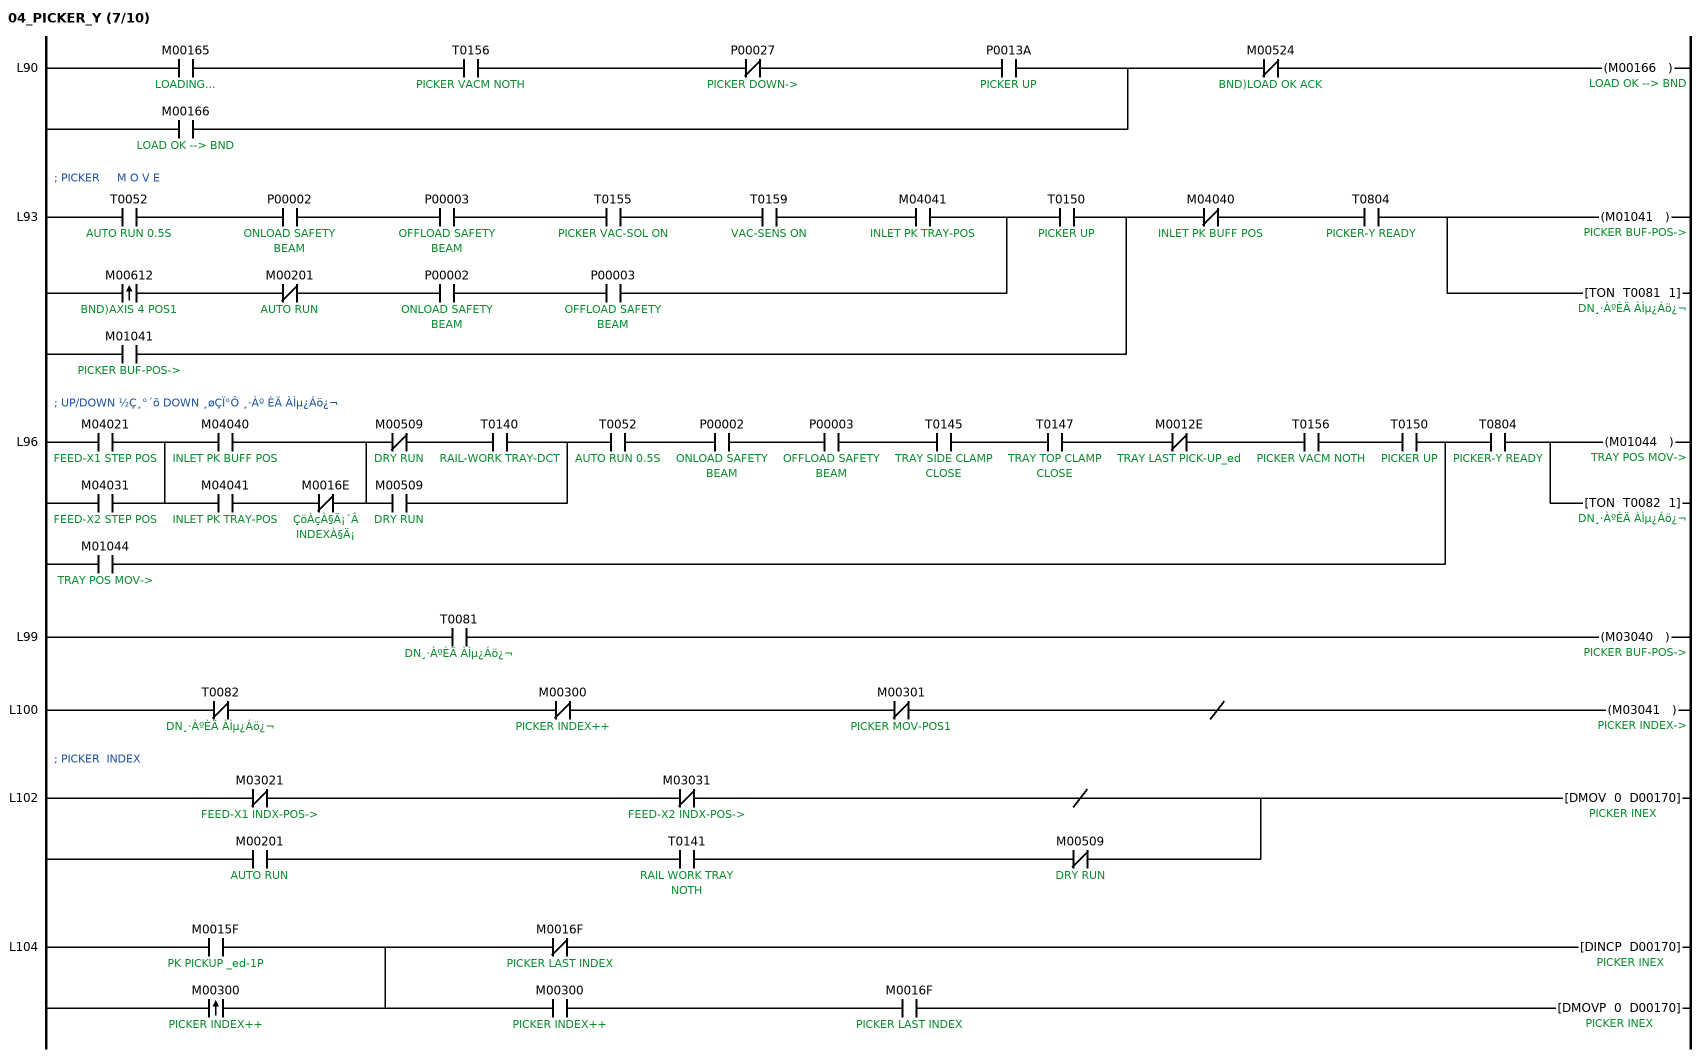
; L90
LOAD      M00165	// LOADING...
AND       T0156	// PICKER VACM NOTH
AND NOT   P00027	// PICKER DOWN->
AND       P0013A	// PICKER UP
OR        M00166	// LOAD OK --> BND
AND NOT   M00524	// BND)LOAD OK ACK
OUT       M00166	// LOAD OK --> BND
// PICKER     M O V E
; L93
LOAD      T0052	// AUTO RUN 0.5S
AND       P00002	// ONLOAD SAFETY BEAM
AND       P00003	// OFFLOAD SAFETY BEAM
AND       T0155	// PICKER VAC-SOL ON
AND       T0159	// VAC-SENS ON
AND       M04041	// INLET PK TRAY-POS
LOADP     M00612	// BND)AXIS 4 POS1
AND NOT   M00201	// AUTO RUN
AND       P00002	// ONLOAD SAFETY BEAM
AND       P00003	// OFFLOAD SAFETY BEAM
OR LOAD
AND       T0150	// PICKER UP
OR        M01041	// PICKER BUF-POS->
AND NOT   M04040	// INLET PK BUFF POS
AND       T0804	// PICKER-Y READY
OUT       M01041	// PICKER BUF-POS->
TON       T0081 1	// DN¸·ÀºÈÄ ÀÌµ¿Áö¿¬
; L96
LOAD      M04021	// FEED-X1 STEP POS
OR        M04031	// FEED-X2 STEP POS
LOAD      M04040	// INLET PK BUFF POS
LOAD      M04041	// INLET PK TRAY-POS
AND NOT   M0016E	// ÇöÀçÀ§Ä¡´Â INDEXÀ§Ä¡
OR LOAD
AND LOAD
LOAD NOT  M00509	// DRY RUN
AND       T0140	// RAIL-WORK TRAY-DCT
OR        M00509	// DRY RUN
AND LOAD
AND       T0052	// AUTO RUN 0.5S
AND       P00002	// ONLOAD SAFETY BEAM
AND       P00003	// OFFLOAD SAFETY BEAM
AND       T0145	// TRAY SIDE CLAMP CLOSE
AND       T0147	// TRAY TOP CLAMP CLOSE
AND NOT   M0012E	// TRAY LAST PICK-UP_ed
AND       T0156	// PICKER VACM NOTH
AND       T0150	// PICKER UP
OR        M01044	// TRAY POS MOV->
AND       T0804	// PICKER-Y READY
OUT       M01044	// TRAY POS MOV->
TON       T0082 1	// DN¸·ÀºÈÄ ÀÌµ¿Áö¿¬
// output comment: UP/DOWN ½Ç¸°´õ DOWN ¸øÇÏ°Ô ¸·Àº ÈÄ ÀÌµ¿Áö¿¬
; L99
LOAD      T0081	// DN¸·ÀºÈÄ ÀÌµ¿Áö¿¬
OUT       M03040	// PICKER BUF-POS->
; L100
LOAD NOT  T0082	// DN¸·ÀºÈÄ ÀÌµ¿Áö¿¬
AND NOT   M00300	// PICKER INDEX++
AND NOT   M00301	// PICKER MOV-POS1
NOT
OUT       M03041	// PICKER INDEX->
// PICKER  INDEX
; L102
LOAD NOT  M03021	// FEED-X1 INDX-POS->
AND NOT   M03031	// FEED-X2 INDX-POS->
NOT
LOAD      M00201	// AUTO RUN
AND       T0141	// RAIL WORK TRAY NOTH
AND NOT   M00509	// DRY RUN
OR LOAD
DMOV      0 D00170	// PICKER INEX
; L104
LOAD      M0015F	// PK PICKUP _ed-1P
ORP       M00300	// PICKER INDEX++
MPUSH
AND NOT   M0016F	// PICKER LAST INDEX
DINCP     D00170	// PICKER INEX
MPOP
AND       M00300	// PICKER INDEX++
AND       M0016F	// PICKER LAST INDEX
DMOVP     0 D00170	// PICKER INEX

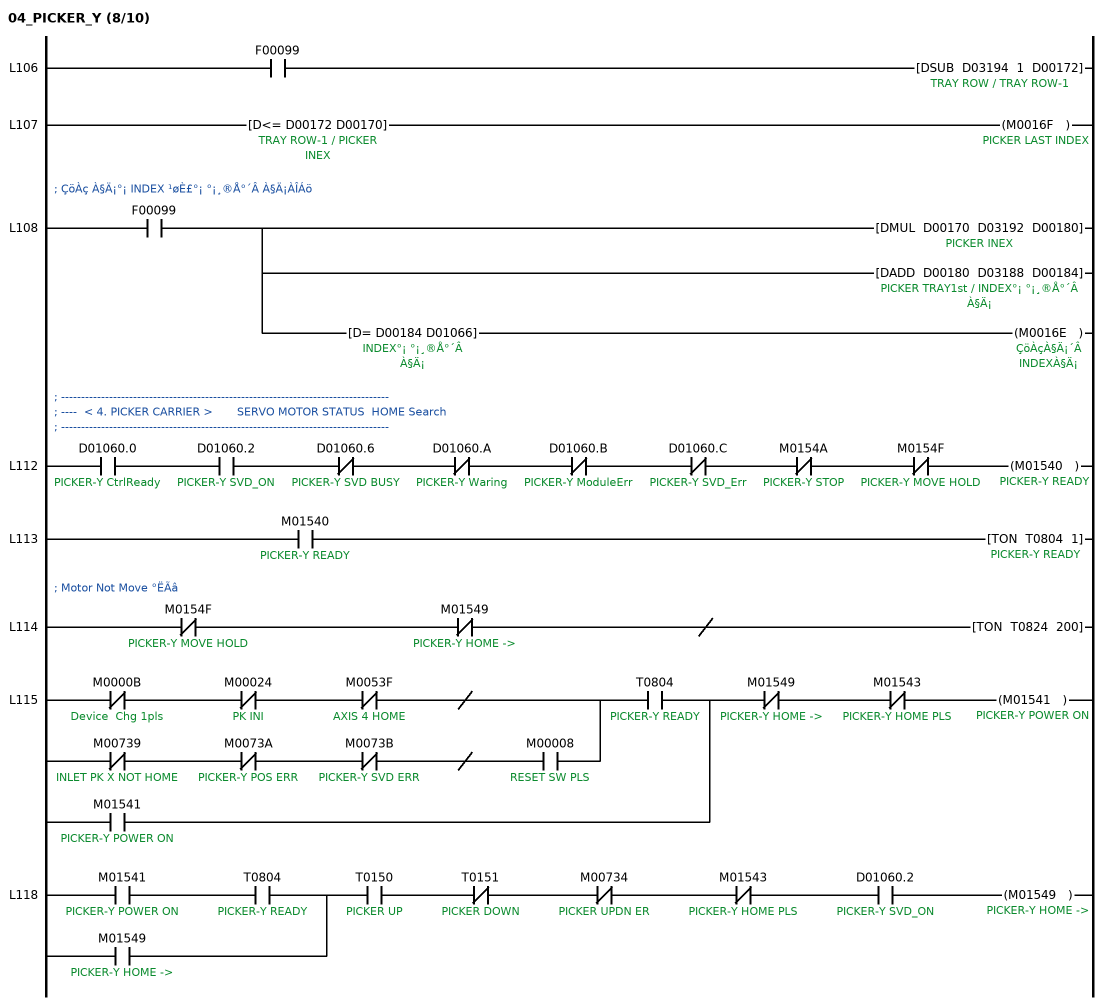
; L106
LOAD      F00099
DSUB      D03194 1 D00172	// TRAY ROW / TRAY ROW-1
; L107
LOADD<=   D00172 D00170	// TRAY ROW-1 / PICKER INEX
OUT       M0016F	// PICKER LAST INDEX
; L108
LOAD      F00099
DMUL      D00170 D03192 D00180	// PICKER INEX
DADD      D00180 D03188 D00184	// PICKER TRAY1st / INDEX°¡ °¡¸®Å°´Â À§Ä¡
ANDD=     D00184 D01066	// INDEX°¡ °¡¸®Å°´Â À§Ä¡
OUT       M0016E	// ÇöÀçÀ§Ä¡´Â INDEXÀ§Ä¡
// output comment: ÇöÀç À§Ä¡°¡ INDEX ¹øÈ£°¡ °¡¸®Å°´Â À§Ä¡ÀÎÁö
// ----------------------------------------------------------------------------------
// 
// ----  < 4. PICKER CARRIER >       SERVO MOTOR STATUS  HOME Search
// 
// ----------------------------------------------------------------------------------
; L112
LOAD      D01060.0	// PICKER-Y CtrlReady
AND       D01060.2	// PICKER-Y SVD_ON
AND NOT   D01060.6	// PICKER-Y SVD BUSY
AND NOT   D01060.A	// PICKER-Y Waring
AND NOT   D01060.B	// PICKER-Y ModuleErr
AND NOT   D01060.C	// PICKER-Y SVD_Err
AND NOT   M0154A	// PICKER-Y STOP
AND NOT   M0154F	// PICKER-Y MOVE HOLD
OUT       M01540	// PICKER-Y READY
; L113
LOAD      M01540	// PICKER-Y READY
TON       T0804 1	// PICKER-Y READY
; L114
LOAD NOT  M0154F	// PICKER-Y MOVE HOLD
AND NOT   M01549	// PICKER-Y HOME ->
NOT
TON       T0824 200
// output comment: Motor Not Move °ËÃâ
; L115
LOAD NOT  M0000B	// Device  Chg 1pls
AND NOT   M00024	// PK INI
AND NOT   M0053F	// AXIS 4 HOME
NOT
LOAD NOT  M00739	// INLET PK X NOT HOME
AND NOT   M0073A	// PICKER-Y POS ERR
AND NOT   M0073B	// PICKER-Y SVD ERR
NOT
AND       M00008	// RESET SW PLS
OR LOAD
AND       T0804	// PICKER-Y READY
OR        M01541	// PICKER-Y POWER ON
AND NOT   M01549	// PICKER-Y HOME ->
AND NOT   M01543	// PICKER-Y HOME PLS
OUT       M01541	// PICKER-Y POWER ON
; L118
LOAD      M01541	// PICKER-Y POWER ON
AND       T0804	// PICKER-Y READY
OR        M01549	// PICKER-Y HOME ->
AND       T0150	// PICKER UP
AND NOT   T0151	// PICKER DOWN
AND NOT   M00734	// PICKER UPDN ER
AND NOT   M01543	// PICKER-Y HOME PLS
AND       D01060.2	// PICKER-Y SVD_ON
OUT       M01549	// PICKER-Y HOME ->

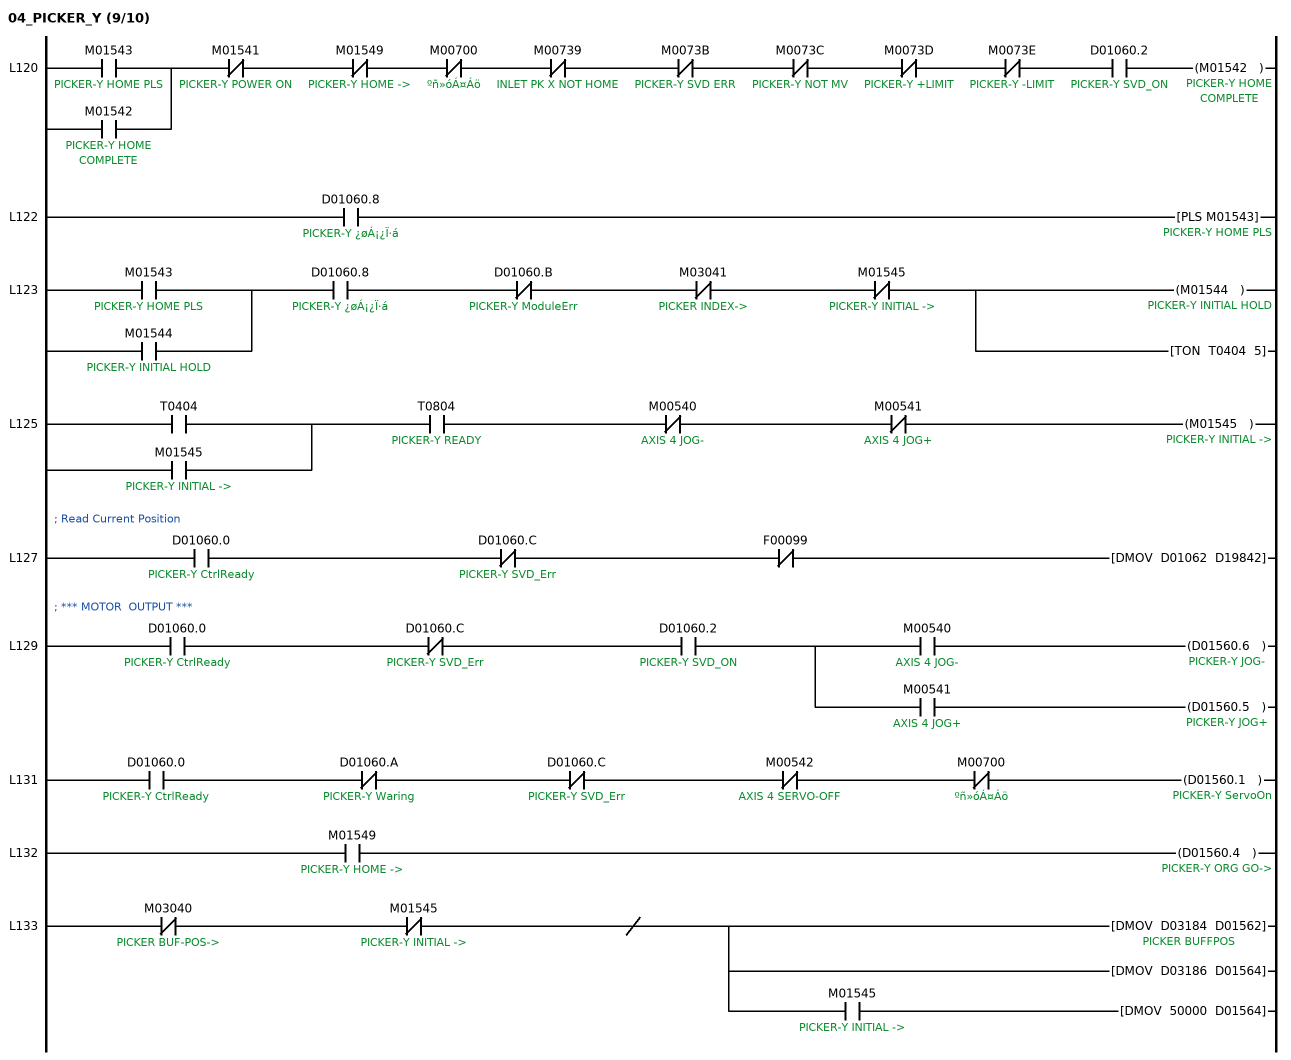
; L120
LOAD      M01543	// PICKER-Y HOME PLS
OR        M01542	// PICKER-Y HOME COMPLETE
AND NOT   M01541	// PICKER-Y POWER ON
AND NOT   M01549	// PICKER-Y HOME ->
AND NOT   M00700	// ºñ»óÁ¤Áö
AND NOT   M00739	// INLET PK X NOT HOME
AND NOT   M0073B	// PICKER-Y SVD ERR
AND NOT   M0073C	// PICKER-Y NOT MV
AND NOT   M0073D	// PICKER-Y +LIMIT
AND NOT   M0073E	// PICKER-Y -LIMIT
AND       D01060.2	// PICKER-Y SVD_ON
OUT       M01542	// PICKER-Y HOME COMPLETE
; L122
LOAD      D01060.8	// PICKER-Y ¿øÁ¡¿Ï·á
OUTP      M01543	// PICKER-Y HOME PLS
; L123
LOAD      M01543	// PICKER-Y HOME PLS
OR        M01544	// PICKER-Y INITIAL HOLD
AND       D01060.8	// PICKER-Y ¿øÁ¡¿Ï·á
AND NOT   D01060.B	// PICKER-Y ModuleErr
AND NOT   M03041	// PICKER INDEX->
AND NOT   M01545	// PICKER-Y INITIAL ->
OUT       M01544	// PICKER-Y INITIAL HOLD
TON       T0404 5
; L125
LOAD      T0404
OR        M01545	// PICKER-Y INITIAL ->
AND       T0804	// PICKER-Y READY
AND NOT   M00540	// AXIS 4 JOG-
AND NOT   M00541	// AXIS 4 JOG+
OUT       M01545	// PICKER-Y INITIAL ->
; L127
LOAD      D01060.0	// PICKER-Y CtrlReady
AND NOT   D01060.C	// PICKER-Y SVD_Err
AND NOT   F00099
DMOV      D01062 D19842
// output comment: Read Current Position
// *** MOTOR  OUTPUT ***
; L129
LOAD      D01060.0	// PICKER-Y CtrlReady
AND NOT   D01060.C	// PICKER-Y SVD_Err
AND       D01060.2	// PICKER-Y SVD_ON
MPUSH
AND       M00540	// AXIS 4 JOG-
OUT       D01560.6	// PICKER-Y JOG-
MPOP
AND       M00541	// AXIS 4 JOG+
OUT       D01560.5	// PICKER-Y JOG+
; L131
LOAD      D01060.0	// PICKER-Y CtrlReady
AND NOT   D01060.A	// PICKER-Y Waring
AND NOT   D01060.C	// PICKER-Y SVD_Err
AND NOT   M00542	// AXIS 4 SERVO-OFF
AND NOT   M00700	// ºñ»óÁ¤Áö
OUT       D01560.1	// PICKER-Y ServoOn
; L132
LOAD      M01549	// PICKER-Y HOME ->
OUT       D01560.4	// PICKER-Y ORG GO->
; L133
LOAD NOT  M03040	// PICKER BUF-POS->
AND NOT   M01545	// PICKER-Y INITIAL ->
NOT
DMOV      D03184 D01562	// PICKER BUFFPOS
DMOV      D03186 D01564
AND       M01545	// PICKER-Y INITIAL ->
DMOV      50000 D01564

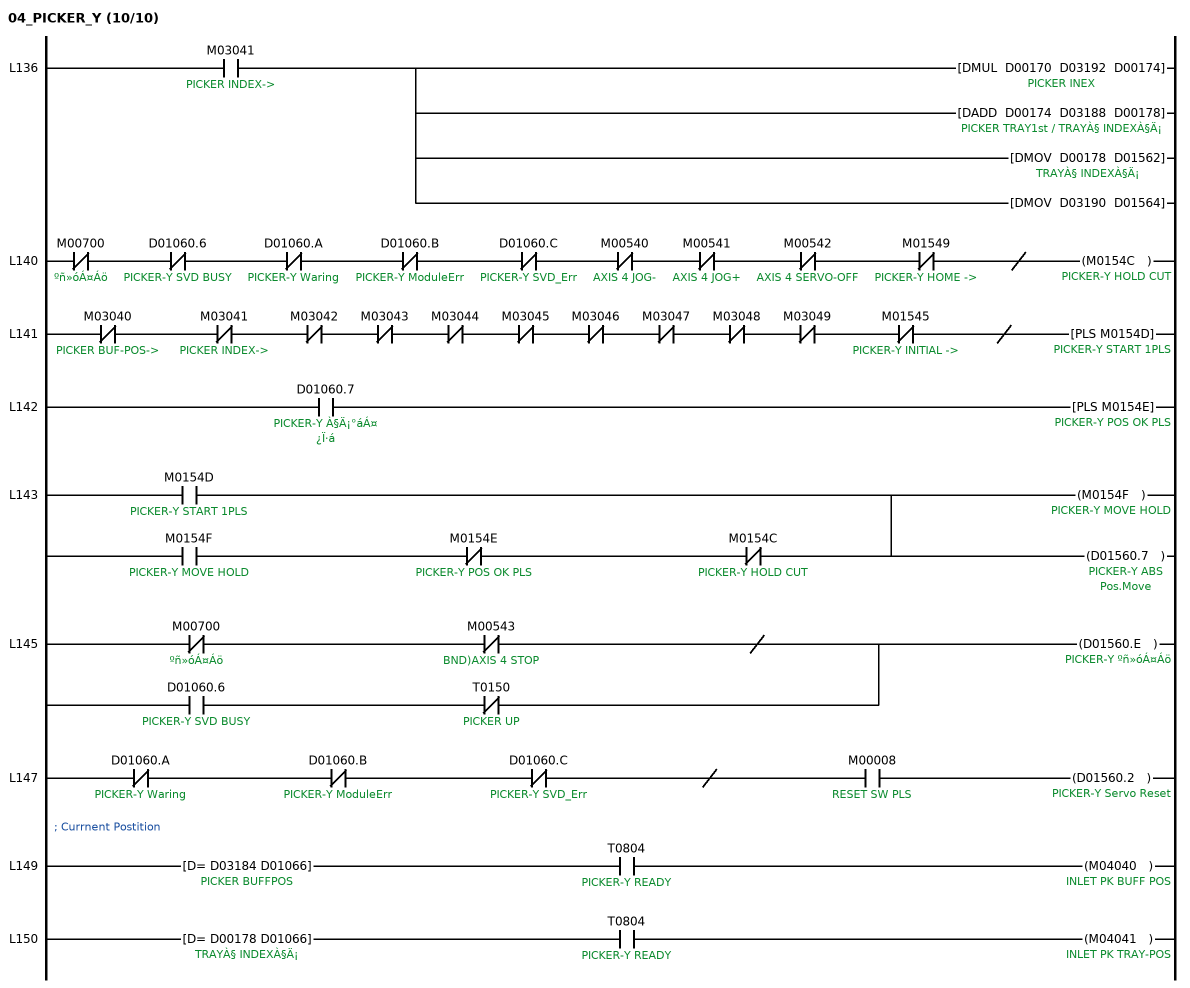
; L136
LOAD      M03041	// PICKER INDEX->
DMUL      D00170 D03192 D00174	// PICKER INEX
DADD      D00174 D03188 D00178	// PICKER TRAY1st / TRAYÀ§ INDEXÀ§Ä¡
DMOV      D00178 D01562	// TRAYÀ§ INDEXÀ§Ä¡
DMOV      D03190 D01564
; L140
LOAD NOT  M00700	// ºñ»óÁ¤Áö
AND NOT   D01060.6	// PICKER-Y SVD BUSY
AND NOT   D01060.A	// PICKER-Y Waring
AND NOT   D01060.B	// PICKER-Y ModuleErr
AND NOT   D01060.C	// PICKER-Y SVD_Err
AND NOT   M00540	// AXIS 4 JOG-
AND NOT   M00541	// AXIS 4 JOG+
AND NOT   M00542	// AXIS 4 SERVO-OFF
AND NOT   M01549	// PICKER-Y HOME ->
NOT
OUT       M0154C	// PICKER-Y HOLD CUT
; L141
LOAD NOT  M03040	// PICKER BUF-POS->
AND NOT   M03041	// PICKER INDEX->
AND NOT   M03042
AND NOT   M03043
AND NOT   M03044
AND NOT   M03045
AND NOT   M03046
AND NOT   M03047
AND NOT   M03048
AND NOT   M03049
AND NOT   M01545	// PICKER-Y INITIAL ->
NOT
OUTP      M0154D	// PICKER-Y START 1PLS
; L142
LOAD      D01060.7	// PICKER-Y À§Ä¡°áÁ¤ ¿Ï·á
OUTP      M0154E	// PICKER-Y POS OK PLS
; L143
LOAD      M0154D	// PICKER-Y START 1PLS
LOAD      M0154F	// PICKER-Y MOVE HOLD
AND NOT   M0154E	// PICKER-Y POS OK PLS
AND NOT   M0154C	// PICKER-Y HOLD CUT
OR LOAD
OUT       M0154F	// PICKER-Y MOVE HOLD
OUT       D01560.7	// PICKER-Y ABS Pos.Move
; L145
LOAD NOT  M00700	// ºñ»óÁ¤Áö
AND NOT   M00543	// BND)AXIS 4 STOP
NOT
LOAD      D01060.6	// PICKER-Y SVD BUSY
AND NOT   T0150	// PICKER UP
OR LOAD
OUT       D01560.E	// PICKER-Y ºñ»óÁ¤Áö
; L147
LOAD NOT  D01060.A	// PICKER-Y Waring
AND NOT   D01060.B	// PICKER-Y ModuleErr
AND NOT   D01060.C	// PICKER-Y SVD_Err
NOT
AND       M00008	// RESET SW PLS
OUT       D01560.2	// PICKER-Y Servo Reset
// Currnent Postition
; L149
LOADD=    D03184 D01066	// PICKER BUFFPOS
AND       T0804	// PICKER-Y READY
OUT       M04040	// INLET PK BUFF POS
; L150
LOADD=    D00178 D01066	// TRAYÀ§ INDEXÀ§Ä¡
AND       T0804	// PICKER-Y READY
OUT       M04041	// INLET PK TRAY-POS

PROGRAM MANUAL (task: ½ºÄµ ÇÁ·Î±×·¥)

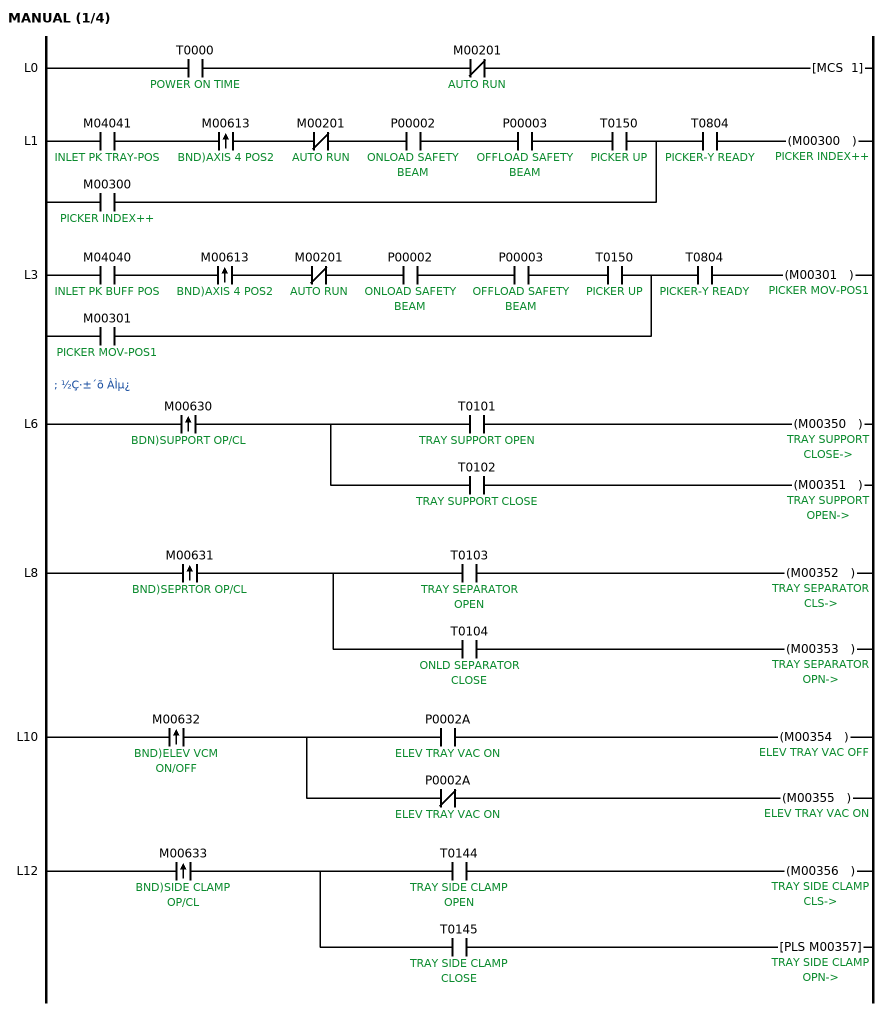
; L0
LOAD      T0000	// POWER ON TIME
AND NOT   M00201	// AUTO RUN
MCS       1
; L1
LOAD      M04041	// INLET PK TRAY-POS
ANDP      M00613	// BND)AXIS 4 POS2
AND NOT   M00201	// AUTO RUN
AND       P00002	// ONLOAD SAFETY BEAM
AND       P00003	// OFFLOAD SAFETY BEAM
AND       T0150	// PICKER UP
OR        M00300	// PICKER INDEX++
AND       T0804	// PICKER-Y READY
OUT       M00300	// PICKER INDEX++
; L3
LOAD      M04040	// INLET PK BUFF POS
ANDP      M00613	// BND)AXIS 4 POS2
AND NOT   M00201	// AUTO RUN
AND       P00002	// ONLOAD SAFETY BEAM
AND       P00003	// OFFLOAD SAFETY BEAM
AND       T0150	// PICKER UP
OR        M00301	// PICKER MOV-POS1
AND       T0804	// PICKER-Y READY
OUT       M00301	// PICKER MOV-POS1
// ½Ç·±´õ ÀÌµ¿
; L6
LOADP     M00630	// BDN)SUPPORT OP/CL
MPUSH
AND       T0101	// TRAY SUPPORT OPEN
OUT       M00350	// TRAY SUPPORT CLOSE->
MPOP
AND       T0102	// TRAY SUPPORT CLOSE
OUT       M00351	// TRAY SUPPORT OPEN->
; L8
LOADP     M00631	// BND)SEPRTOR OP/CL
MPUSH
AND       T0103	// TRAY SEPARATOR OPEN
OUT       M00352	// TRAY SEPARATOR CLS->
MPOP
AND       T0104	// ONLD SEPARATOR CLOSE
OUT       M00353	// TRAY SEPARATOR OPN->
; L10
LOADP     M00632	// BND)ELEV VCM ON/OFF
MPUSH
AND       P0002A	// ELEV TRAY VAC ON
OUT       M00354	// ELEV TRAY VAC OFF
MPOP
AND NOT   P0002A	// ELEV TRAY VAC ON
OUT       M00355	// ELEV TRAY VAC ON
; L12
LOADP     M00633	// BND)SIDE CLAMP OP/CL
MPUSH
AND       T0144	// TRAY SIDE CLAMP OPEN
OUT       M00356	// TRAY SIDE CLAMP CLS->
MPOP
AND       T0145	// TRAY SIDE CLAMP CLOSE
OUTP      M00357	// TRAY SIDE CLAMP OPN->

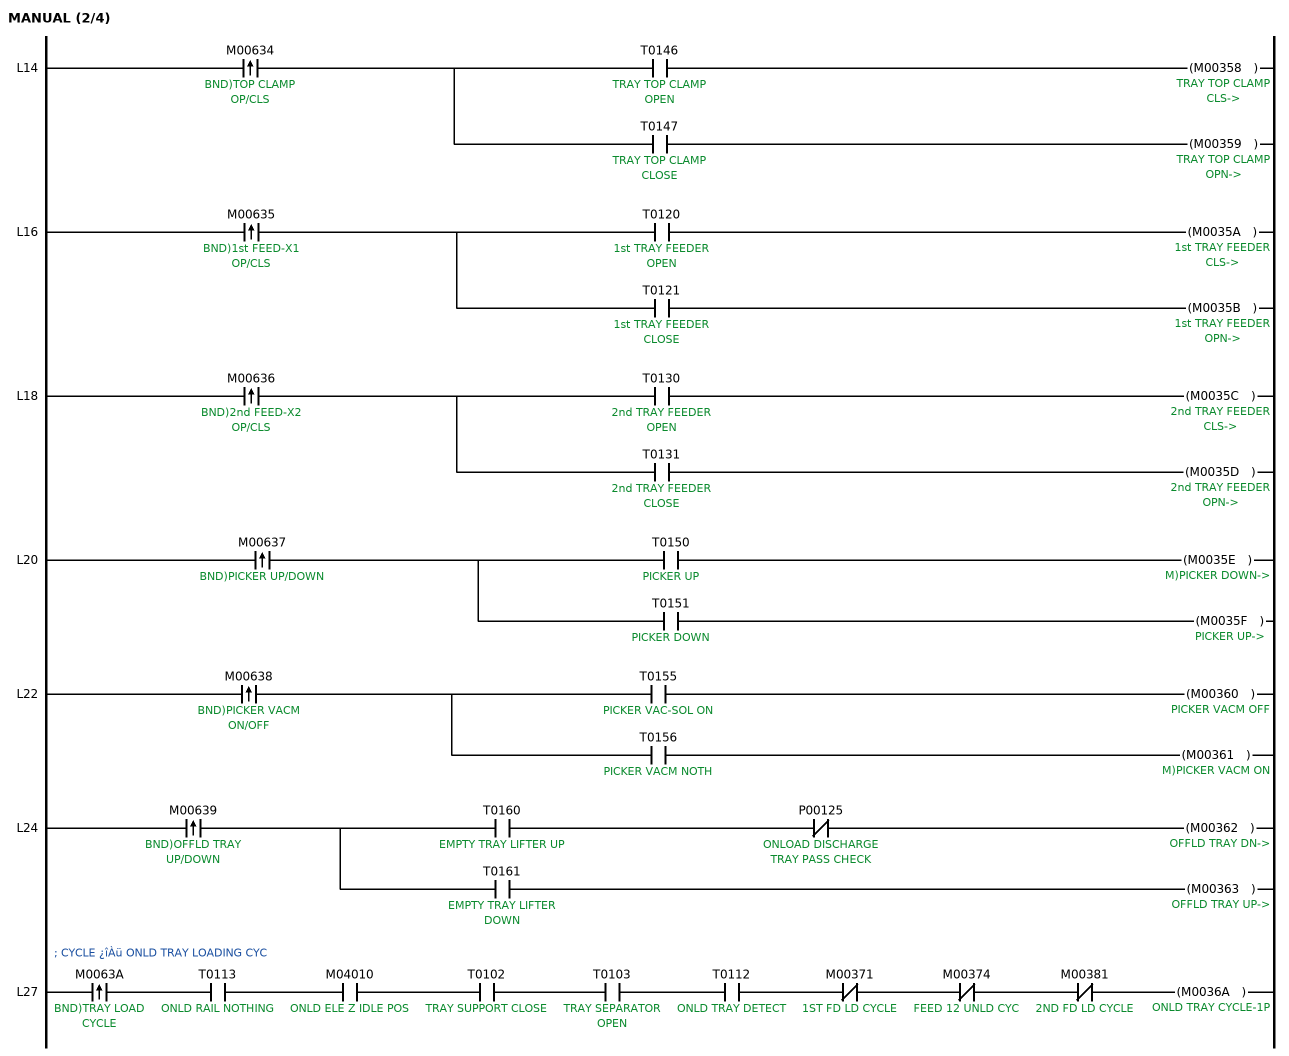
; L14
LOADP     M00634	// BND)TOP CLAMP OP/CLS
MPUSH
AND       T0146	// TRAY TOP CLAMP OPEN
OUT       M00358	// TRAY TOP CLAMP CLS->
MPOP
AND       T0147	// TRAY TOP CLAMP CLOSE
OUT       M00359	// TRAY TOP CLAMP OPN->
; L16
LOADP     M00635	// BND)1st FEED-X1 OP/CLS
MPUSH
AND       T0120	// 1st TRAY FEEDER OPEN
OUT       M0035A	// 1st TRAY FEEDER CLS->
MPOP
AND       T0121	// 1st TRAY FEEDER CLOSE
OUT       M0035B	// 1st TRAY FEEDER OPN->
; L18
LOADP     M00636	// BND)2nd FEED-X2 OP/CLS
MPUSH
AND       T0130	// 2nd TRAY FEEDER OPEN
OUT       M0035C	// 2nd TRAY FEEDER CLS->
MPOP
AND       T0131	// 2nd TRAY FEEDER CLOSE
OUT       M0035D	// 2nd TRAY FEEDER OPN->
; L20
LOADP     M00637	// BND)PICKER UP/DOWN
MPUSH
AND       T0150	// PICKER UP
OUT       M0035E	// M)PICKER DOWN->
MPOP
AND       T0151	// PICKER DOWN
OUT       M0035F	// PICKER UP->
; L22
LOADP     M00638	// BND)PICKER VACM ON/OFF
MPUSH
AND       T0155	// PICKER VAC-SOL ON
OUT       M00360	// PICKER VACM OFF
MPOP
AND       T0156	// PICKER VACM NOTH
OUT       M00361	// M)PICKER VACM ON
; L24
LOADP     M00639	// BND)OFFLD TRAY UP/DOWN
MPUSH
AND       T0160	// EMPTY TRAY LIFTER UP
AND NOT   P00125	// ONLOAD DISCHARGE TRAY PASS CHECK
OUT       M00362	// OFFLD TRAY DN->
MPOP
AND       T0161	// EMPTY TRAY LIFTER DOWN
OUT       M00363	// OFFLD TRAY UP->
// CYCLE ¿îÀü ONLD TRAY LOADING CYC
; L27
LOADP     M0063A	// BND)TRAY LOAD CYCLE
AND       T0113	// ONLD RAIL NOTHING
AND       M04010	// ONLD ELE Z IDLE POS
AND       T0102	// TRAY SUPPORT CLOSE
AND       T0103	// TRAY SEPARATOR OPEN
AND       T0112	// ONLD TRAY DETECT
AND NOT   M00371	// 1ST FD LD CYCLE
AND NOT   M00374	// FEED 12 UNLD CYC
AND NOT   M00381	// 2ND FD LD CYCLE
OUT       M0036A	// ONLD TRAY CYCLE-1P

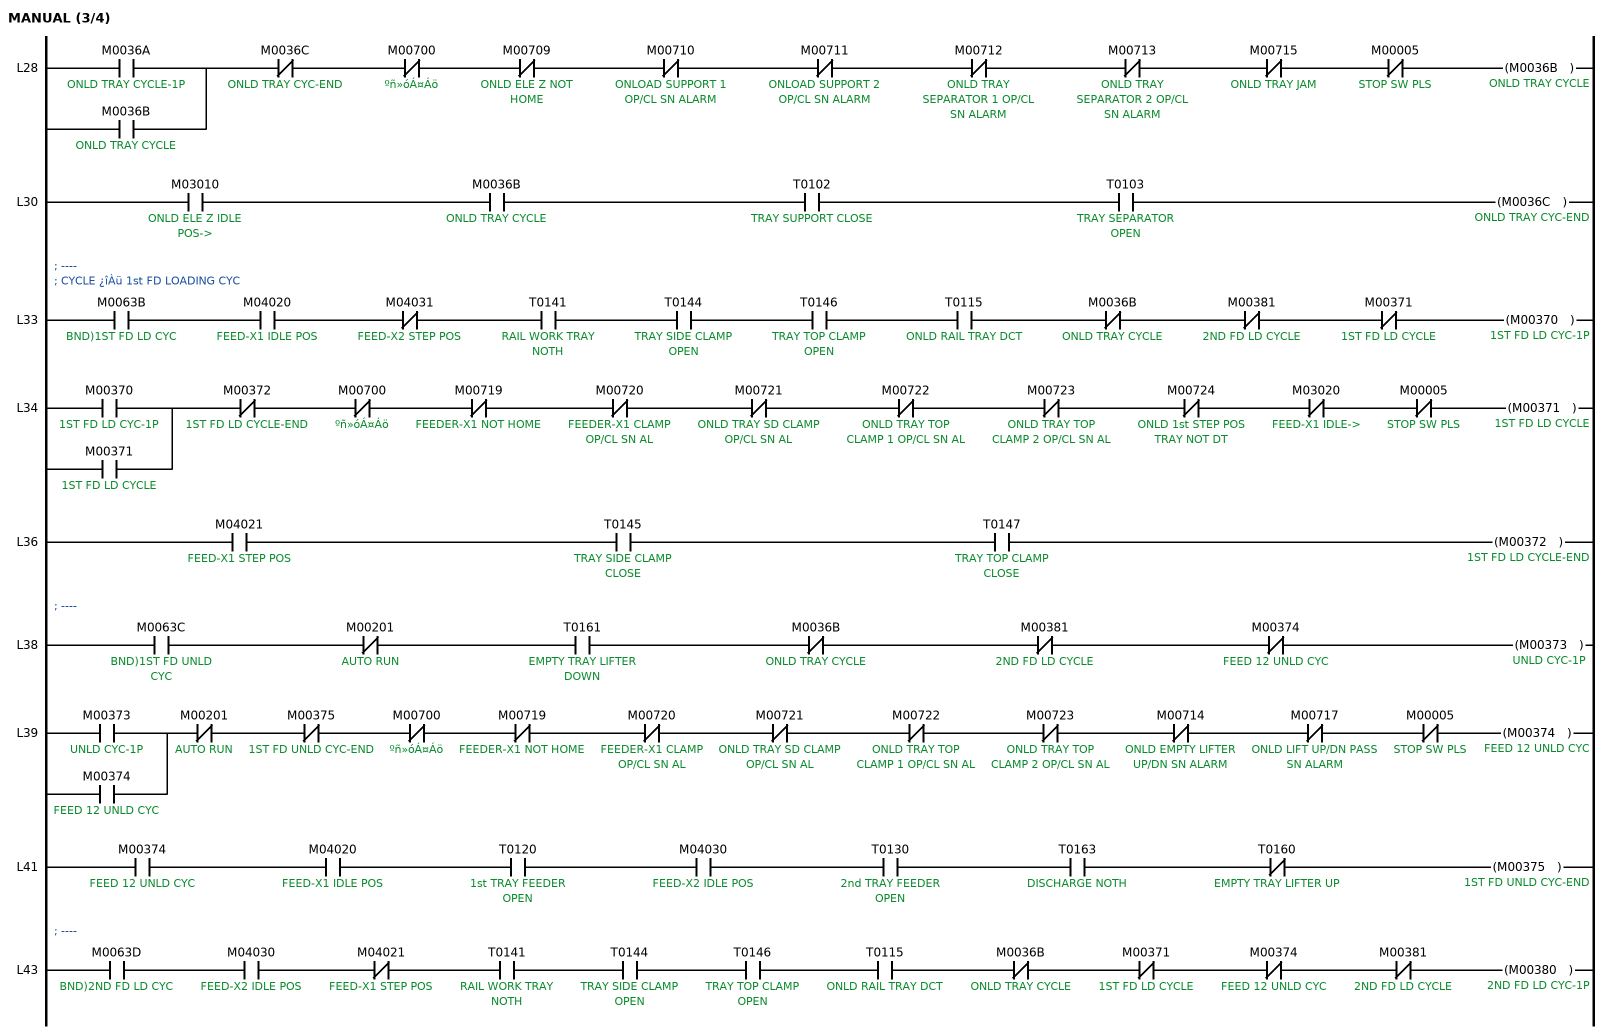
; L28
LOAD      M0036A	// ONLD TRAY CYCLE-1P
OR        M0036B	// ONLD TRAY CYCLE
AND NOT   M0036C	// ONLD TRAY CYC-END
AND NOT   M00700	// ºñ»óÁ¤Áö
AND NOT   M00709	// ONLD ELE Z NOT HOME
AND NOT   M00710	// ONLOAD SUPPORT 1 OP/CL SN ALARM
AND NOT   M00711	// ONLOAD SUPPORT 2 OP/CL SN ALARM
AND NOT   M00712	// ONLD TRAY SEPARATOR 1 OP/CL SN ALARM
AND NOT   M00713	// ONLD TRAY SEPARATOR 2 OP/CL SN ALARM
AND NOT   M00715	// ONLD TRAY JAM
AND NOT   M00005	// STOP SW PLS
OUT       M0036B	// ONLD TRAY CYCLE
; L30
LOAD      M03010	// ONLD ELE Z IDLE POS->
AND       M0036B	// ONLD TRAY CYCLE
AND       T0102	// TRAY SUPPORT CLOSE
AND       T0103	// TRAY SEPARATOR OPEN
OUT       M0036C	// ONLD TRAY CYC-END
// ----
// CYCLE ¿îÀü 1st FD LOADING CYC
; L33
LOAD      M0063B	// BND)1ST FD LD CYC
AND       M04020	// FEED-X1 IDLE POS
AND NOT   M04031	// FEED-X2 STEP POS
AND       T0141	// RAIL WORK TRAY NOTH
AND       T0144	// TRAY SIDE CLAMP OPEN
AND       T0146	// TRAY TOP CLAMP OPEN
AND       T0115	// ONLD RAIL TRAY DCT
AND NOT   M0036B	// ONLD TRAY CYCLE
AND NOT   M00381	// 2ND FD LD CYCLE
AND NOT   M00371	// 1ST FD LD CYCLE
OUT       M00370	// 1ST FD LD CYC-1P
; L34
LOAD      M00370	// 1ST FD LD CYC-1P
OR        M00371	// 1ST FD LD CYCLE
AND NOT   M00372	// 1ST FD LD CYCLE-END
AND NOT   M00700	// ºñ»óÁ¤Áö
AND NOT   M00719	// FEEDER-X1 NOT HOME
AND NOT   M00720	// FEEDER-X1 CLAMP OP/CL SN AL
AND NOT   M00721	// ONLD TRAY SD CLAMP OP/CL SN AL
AND NOT   M00722	// ONLD TRAY TOP CLAMP 1 OP/CL SN AL
AND NOT   M00723	// ONLD TRAY TOP CLAMP 2 OP/CL SN AL
AND NOT   M00724	// ONLD 1st STEP POS TRAY NOT DT
AND NOT   M03020	// FEED-X1 IDLE->
AND NOT   M00005	// STOP SW PLS
OUT       M00371	// 1ST FD LD CYCLE
; L36
LOAD      M04021	// FEED-X1 STEP POS
AND       T0145	// TRAY SIDE CLAMP CLOSE
AND       T0147	// TRAY TOP CLAMP CLOSE
OUT       M00372	// 1ST FD LD CYCLE-END
// ----
; L38
LOAD      M0063C	// BND)1ST FD UNLD CYC
AND NOT   M00201	// AUTO RUN
AND       T0161	// EMPTY TRAY LIFTER DOWN
AND NOT   M0036B	// ONLD TRAY CYCLE
AND NOT   M00381	// 2ND FD LD CYCLE
AND NOT   M00374	// FEED 12 UNLD CYC
OUT       M00373	// UNLD CYC-1P
; L39
LOAD      M00373	// UNLD CYC-1P
OR        M00374	// FEED 12 UNLD CYC
AND NOT   M00201	// AUTO RUN
AND NOT   M00375	// 1ST FD UNLD CYC-END
AND NOT   M00700	// ºñ»óÁ¤Áö
AND NOT   M00719	// FEEDER-X1 NOT HOME
AND NOT   M00720	// FEEDER-X1 CLAMP OP/CL SN AL
AND NOT   M00721	// ONLD TRAY SD CLAMP OP/CL SN AL
AND NOT   M00722	// ONLD TRAY TOP CLAMP 1 OP/CL SN AL
AND NOT   M00723	// ONLD TRAY TOP CLAMP 2 OP/CL SN AL
AND NOT   M00714	// ONLD EMPTY LIFTER UP/DN SN ALARM
AND NOT   M00717	// ONLD LIFT UP/DN PASS SN ALARM
AND NOT   M00005	// STOP SW PLS
OUT       M00374	// FEED 12 UNLD CYC
; L41
LOAD      M00374	// FEED 12 UNLD CYC
AND       M04020	// FEED-X1 IDLE POS
AND       T0120	// 1st TRAY FEEDER OPEN
AND       M04030	// FEED-X2 IDLE POS
AND       T0130	// 2nd TRAY FEEDER OPEN
AND       T0163	// DISCHARGE NOTH
AND NOT   T0160	// EMPTY TRAY LIFTER UP
OUT       M00375	// 1ST FD UNLD CYC-END
// ----
; L43
LOAD      M0063D	// BND)2ND FD LD CYC
AND       M04030	// FEED-X2 IDLE POS
AND NOT   M04021	// FEED-X1 STEP POS
AND       T0141	// RAIL WORK TRAY NOTH
AND       T0144	// TRAY SIDE CLAMP OPEN
AND       T0146	// TRAY TOP CLAMP OPEN
AND       T0115	// ONLD RAIL TRAY DCT
AND NOT   M0036B	// ONLD TRAY CYCLE
AND NOT   M00371	// 1ST FD LD CYCLE
AND NOT   M00374	// FEED 12 UNLD CYC
AND NOT   M00381	// 2ND FD LD CYCLE
OUT       M00380	// 2ND FD LD CYC-1P

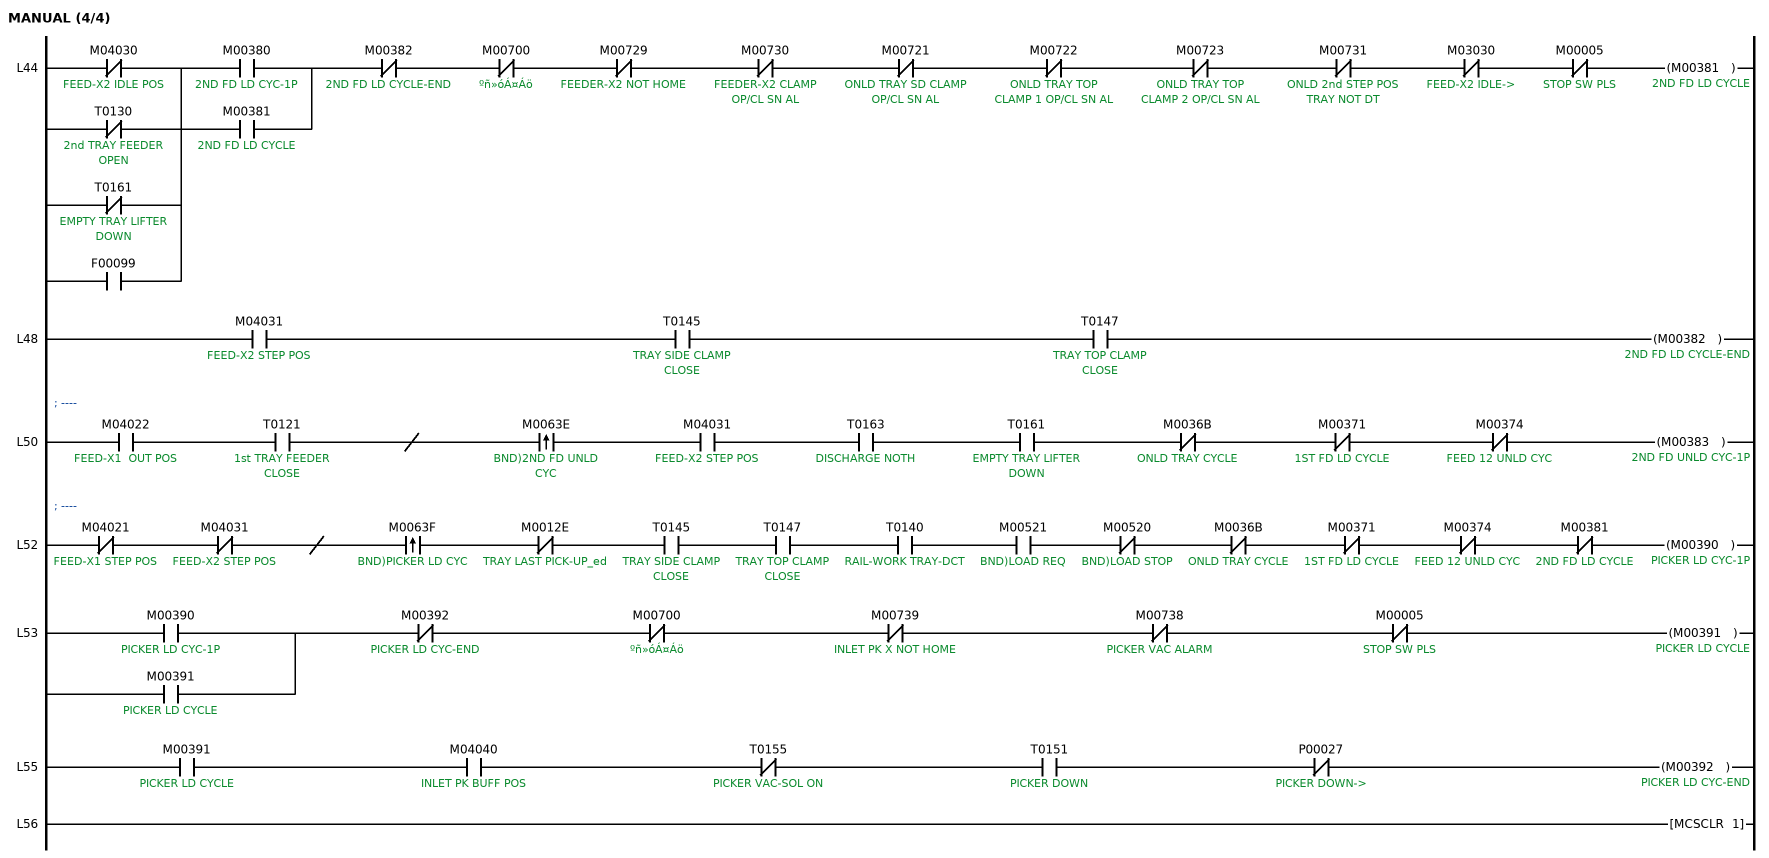
; L44
LOAD NOT  M04030	// FEED-X2 IDLE POS
OR NOT    T0130	// 2nd TRAY FEEDER OPEN
OR NOT    T0161	// EMPTY TRAY LIFTER DOWN
OR        F00099
LOAD      M00380	// 2ND FD LD CYC-1P
OR        M00381	// 2ND FD LD CYCLE
AND LOAD
AND NOT   M00382	// 2ND FD LD CYCLE-END
AND NOT   M00700	// ºñ»óÁ¤Áö
AND NOT   M00729	// FEEDER-X2 NOT HOME
AND NOT   M00730	// FEEDER-X2 CLAMP OP/CL SN AL
AND NOT   M00721	// ONLD TRAY SD CLAMP OP/CL SN AL
AND NOT   M00722	// ONLD TRAY TOP CLAMP 1 OP/CL SN AL
AND NOT   M00723	// ONLD TRAY TOP CLAMP 2 OP/CL SN AL
AND NOT   M00731	// ONLD 2nd STEP POS TRAY NOT DT
AND NOT   M03030	// FEED-X2 IDLE->
AND NOT   M00005	// STOP SW PLS
OUT       M00381	// 2ND FD LD CYCLE
; L48
LOAD      M04031	// FEED-X2 STEP POS
AND       T0145	// TRAY SIDE CLAMP CLOSE
AND       T0147	// TRAY TOP CLAMP CLOSE
OUT       M00382	// 2ND FD LD CYCLE-END
// ----
; L50
LOAD      M04022	// FEED-X1  OUT POS
AND       T0121	// 1st TRAY FEEDER CLOSE
NOT
ANDP      M0063E	// BND)2ND FD UNLD CYC
AND       M04031	// FEED-X2 STEP POS
AND       T0163	// DISCHARGE NOTH
AND       T0161	// EMPTY TRAY LIFTER DOWN
AND NOT   M0036B	// ONLD TRAY CYCLE
AND NOT   M00371	// 1ST FD LD CYCLE
AND NOT   M00374	// FEED 12 UNLD CYC
OUT       M00383	// 2ND FD UNLD CYC-1P
// ----
; L52
LOAD NOT  M04021	// FEED-X1 STEP POS
AND NOT   M04031	// FEED-X2 STEP POS
NOT
ANDP      M0063F	// BND)PICKER LD CYC
AND NOT   M0012E	// TRAY LAST PICK-UP_ed
AND       T0145	// TRAY SIDE CLAMP CLOSE
AND       T0147	// TRAY TOP CLAMP CLOSE
AND       T0140	// RAIL-WORK TRAY-DCT
AND       M00521	// BND)LOAD REQ
AND NOT   M00520	// BND)LOAD STOP
AND NOT   M0036B	// ONLD TRAY CYCLE
AND NOT   M00371	// 1ST FD LD CYCLE
AND NOT   M00374	// FEED 12 UNLD CYC
AND NOT   M00381	// 2ND FD LD CYCLE
OUT       M00390	// PICKER LD CYC-1P
; L53
LOAD      M00390	// PICKER LD CYC-1P
OR        M00391	// PICKER LD CYCLE
AND NOT   M00392	// PICKER LD CYC-END
AND NOT   M00700	// ºñ»óÁ¤Áö
AND NOT   M00739	// INLET PK X NOT HOME
AND NOT   M00738	// PICKER VAC ALARM
AND NOT   M00005	// STOP SW PLS
OUT       M00391	// PICKER LD CYCLE
; L55
LOAD      M00391	// PICKER LD CYCLE
AND       M04040	// INLET PK BUFF POS
AND NOT   T0155	// PICKER VAC-SOL ON
AND       T0151	// PICKER DOWN
AND NOT   P00027	// PICKER DOWN->
OUT       M00392	// PICKER LD CYC-END
; L56
MCSCLR    1

PROGRAM OUTPUT (task: ½ºÄµ ÇÁ·Î±×·¥)

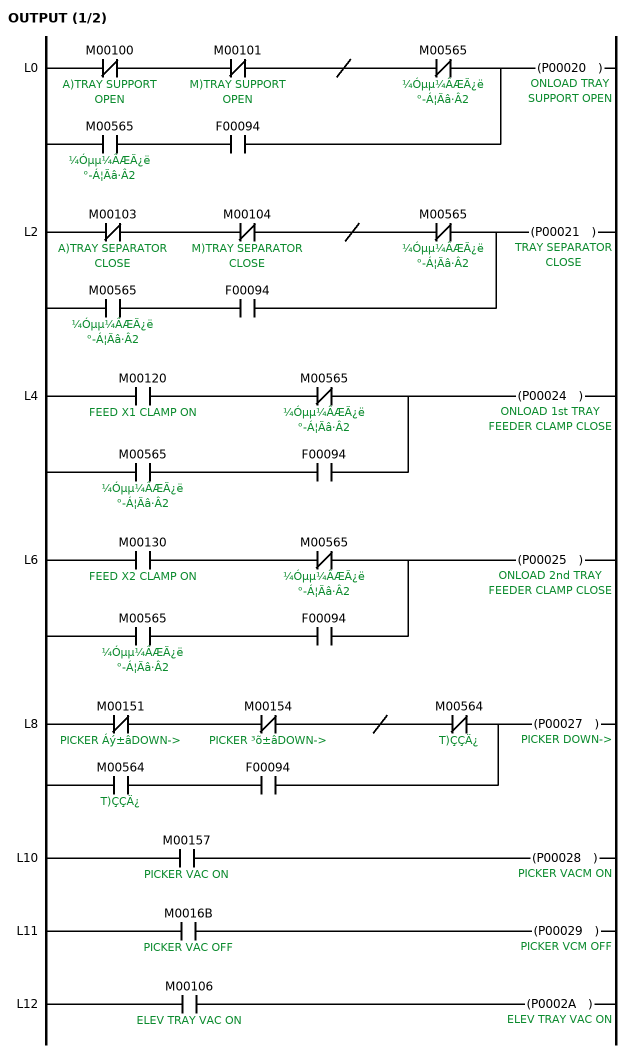
; L0
LOAD NOT  M00100	// A)TRAY SUPPORT OPEN
AND NOT   M00101	// M)TRAY SUPPORT OPEN
NOT
AND NOT   M00565	// ¼Óµµ¼ÂÆÃ¿ë °­Á¦Ãâ·Â2
LOAD      M00565	// ¼Óµµ¼ÂÆÃ¿ë °­Á¦Ãâ·Â2
AND       F00094
OR LOAD
OUT       P00020	// ONLOAD TRAY SUPPORT OPEN
; L2
LOAD NOT  M00103	// A)TRAY SEPARATOR CLOSE
AND NOT   M00104	// M)TRAY SEPARATOR CLOSE
NOT
AND NOT   M00565	// ¼Óµµ¼ÂÆÃ¿ë °­Á¦Ãâ·Â2
LOAD      M00565	// ¼Óµµ¼ÂÆÃ¿ë °­Á¦Ãâ·Â2
AND       F00094
OR LOAD
OUT       P00021	// TRAY SEPARATOR CLOSE
; L4
LOAD      M00120	// FEED X1 CLAMP ON
AND NOT   M00565	// ¼Óµµ¼ÂÆÃ¿ë °­Á¦Ãâ·Â2
LOAD      M00565	// ¼Óµµ¼ÂÆÃ¿ë °­Á¦Ãâ·Â2
AND       F00094
OR LOAD
OUT       P00024	// ONLOAD 1st TRAY FEEDER CLAMP CLOSE
; L6
LOAD      M00130	// FEED X2 CLAMP ON
AND NOT   M00565	// ¼Óµµ¼ÂÆÃ¿ë °­Á¦Ãâ·Â2
LOAD      M00565	// ¼Óµµ¼ÂÆÃ¿ë °­Á¦Ãâ·Â2
AND       F00094
OR LOAD
OUT       P00025	// ONLOAD 2nd TRAY FEEDER CLAMP CLOSE
; L8
LOAD NOT  M00151	// PICKER Áý±âDOWN->
AND NOT   M00154	// PICKER ³õ±âDOWN->
NOT
AND NOT   M00564	// T)ÇÇÄ¿
LOAD      M00564	// T)ÇÇÄ¿
AND       F00094
OR LOAD
OUT       P00027	// PICKER DOWN->
; L10
LOAD      M00157	// PICKER VAC ON
OUT       P00028	// PICKER VACM ON
; L11
LOAD      M0016B	// PICKER VAC OFF
OUT       P00029	// PICKER VCM OFF
; L12
LOAD      M00106	// ELEV TRAY VAC ON
OUT       P0002A	// ELEV TRAY VAC ON

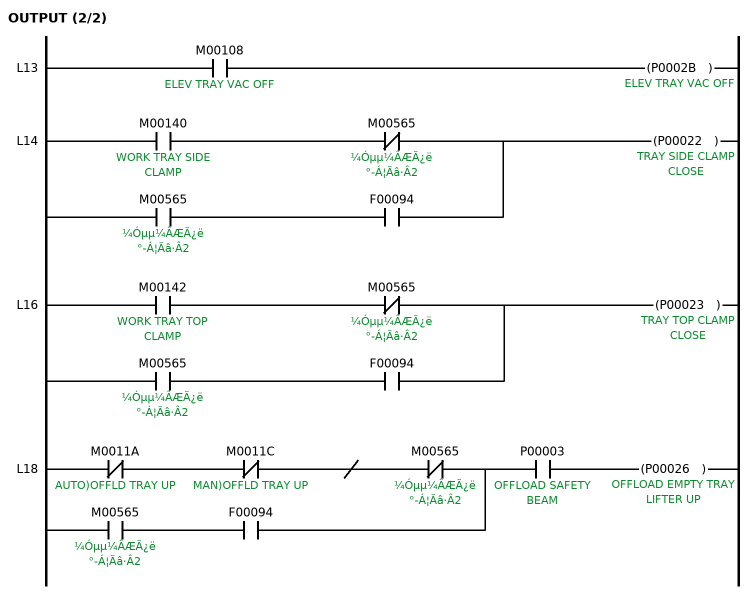
; L13
LOAD      M00108	// ELEV TRAY VAC OFF
OUT       P0002B	// ELEV TRAY VAC OFF
; L14
LOAD      M00140	// WORK TRAY SIDE CLAMP
AND NOT   M00565	// ¼Óµµ¼ÂÆÃ¿ë °­Á¦Ãâ·Â2
LOAD      M00565	// ¼Óµµ¼ÂÆÃ¿ë °­Á¦Ãâ·Â2
AND       F00094
OR LOAD
OUT       P00022	// TRAY SIDE CLAMP CLOSE
; L16
LOAD      M00142	// WORK TRAY TOP CLAMP
AND NOT   M00565	// ¼Óµµ¼ÂÆÃ¿ë °­Á¦Ãâ·Â2
LOAD      M00565	// ¼Óµµ¼ÂÆÃ¿ë °­Á¦Ãâ·Â2
AND       F00094
OR LOAD
OUT       P00023	// TRAY TOP CLAMP CLOSE
; L18
LOAD NOT  M0011A	// AUTO)OFFLD TRAY UP
AND NOT   M0011C	// MAN)OFFLD TRAY UP
NOT
AND NOT   M00565	// ¼Óµµ¼ÂÆÃ¿ë °­Á¦Ãâ·Â2
LOAD      M00565	// ¼Óµµ¼ÂÆÃ¿ë °­Á¦Ãâ·Â2
AND       F00094
OR LOAD
AND       P00003	// OFFLOAD SAFETY BEAM
OUT       P00026	// OFFLOAD EMPTY TRAY LIFTER UP

PROGRAM ALARM (task: ½ºÄµ ÇÁ·Î±×·¥)

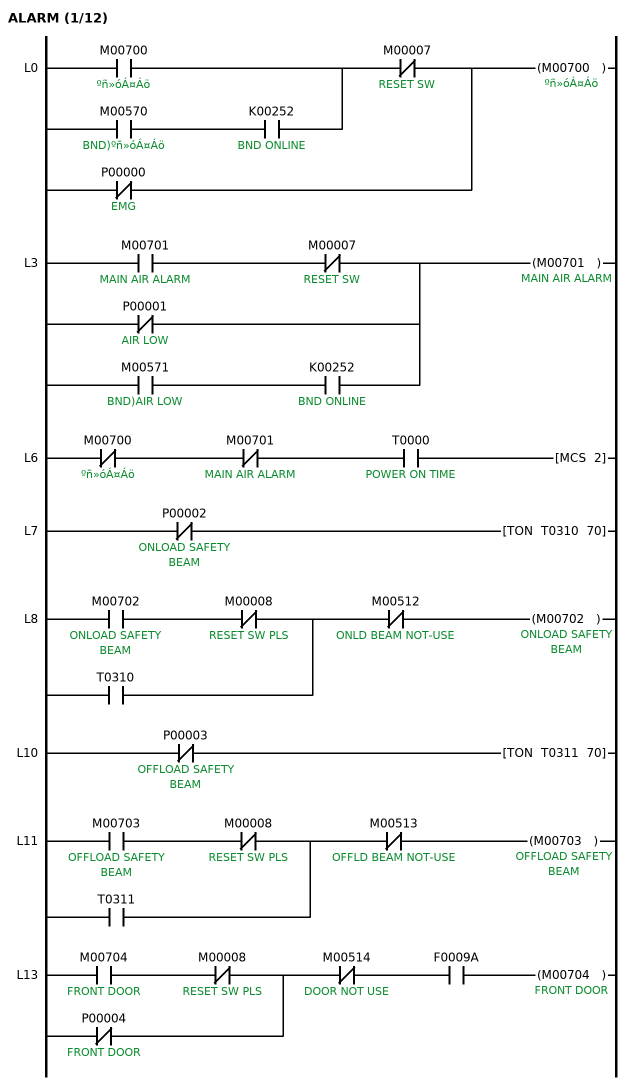
; L0
LOAD      M00700	// ºñ»óÁ¤Áö
LOAD      M00570	// BND)ºñ»óÁ¤Áö
AND       K00252	// BND ONLINE
OR LOAD
AND NOT   M00007	// RESET SW
OR NOT    P00000	// EMG
OUT       M00700	// ºñ»óÁ¤Áö
; L3
LOAD      M00701	// MAIN AIR ALARM
AND NOT   M00007	// RESET SW
OR NOT    P00001	// AIR LOW
LOAD      M00571	// BND)AIR LOW
AND       K00252	// BND ONLINE
OR LOAD
OUT       M00701	// MAIN AIR ALARM
; L6
LOAD NOT  M00700	// ºñ»óÁ¤Áö
AND NOT   M00701	// MAIN AIR ALARM
AND       T0000	// POWER ON TIME
MCS       2
; L7
LOAD NOT  P00002	// ONLOAD SAFETY BEAM
TON       T0310 70
; L8
LOAD      M00702	// ONLOAD SAFETY BEAM
AND NOT   M00008	// RESET SW PLS
OR        T0310
AND NOT   M00512	// ONLD BEAM NOT-USE
OUT       M00702	// ONLOAD SAFETY BEAM
; L10
LOAD NOT  P00003	// OFFLOAD SAFETY BEAM
TON       T0311 70
; L11
LOAD      M00703	// OFFLOAD SAFETY BEAM
AND NOT   M00008	// RESET SW PLS
OR        T0311
AND NOT   M00513	// OFFLD BEAM NOT-USE
OUT       M00703	// OFFLOAD SAFETY BEAM
; L13
LOAD      M00704	// FRONT DOOR
AND NOT   M00008	// RESET SW PLS
OR NOT    P00004	// FRONT DOOR
AND NOT   M00514	// DOOR NOT USE
AND       F0009A
OUT       M00704	// FRONT DOOR

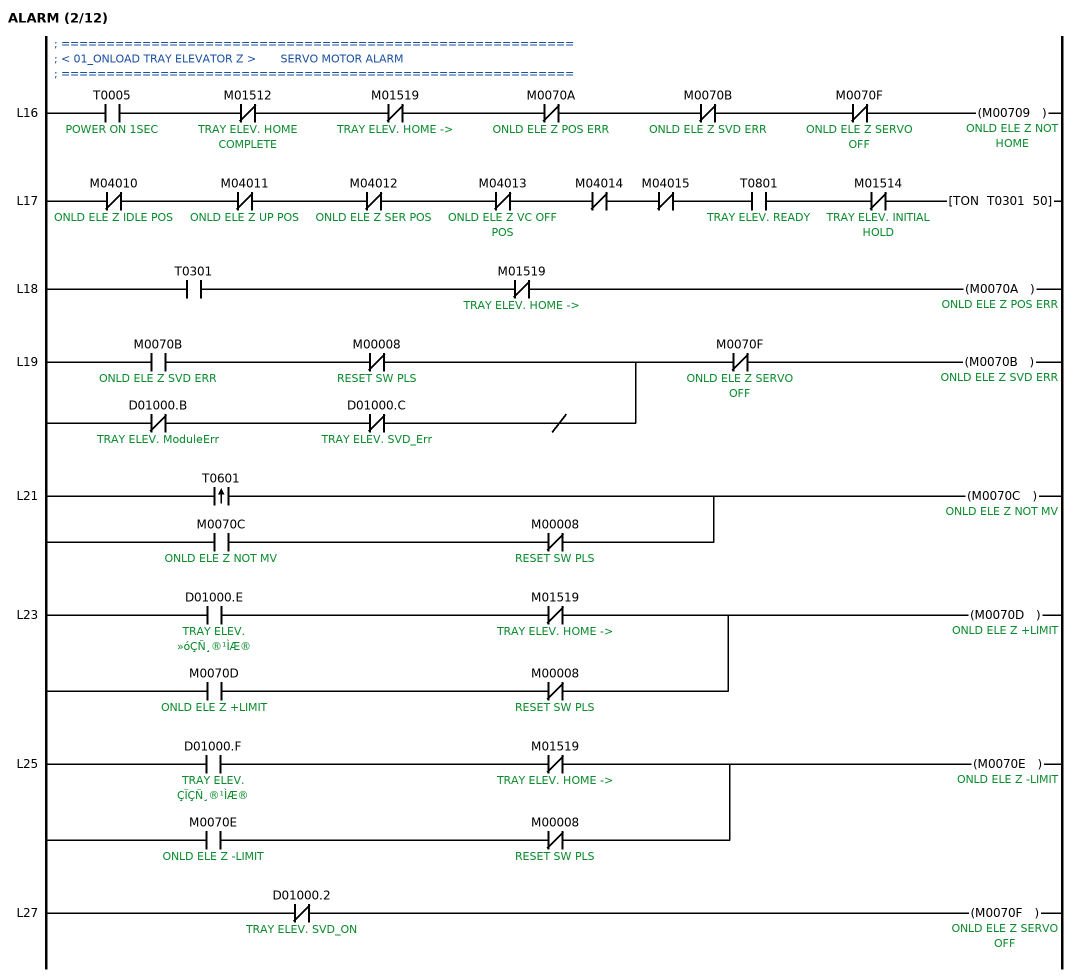
// =========================================================
// 
//        < 01_ONLOAD TRAY ELEVATOR Z >       SERVO MOTOR ALARM
// 
// =========================================================
; L16
LOAD      T0005	// POWER ON 1SEC
AND NOT   M01512	// TRAY ELEV. HOME COMPLETE
AND NOT   M01519	// TRAY ELEV. HOME ->
AND NOT   M0070A	// ONLD ELE Z POS ERR
AND NOT   M0070B	// ONLD ELE Z SVD ERR
AND NOT   M0070F	// ONLD ELE Z SERVO OFF
OUT       M00709	// ONLD ELE Z NOT HOME
; L17
LOAD NOT  M04010	// ONLD ELE Z IDLE POS
AND NOT   M04011	// ONLD ELE Z UP POS
AND NOT   M04012	// ONLD ELE Z SER POS
AND NOT   M04013	// ONLD ELE Z VC OFF POS
AND NOT   M04014
AND NOT   M04015
AND       T0801	// TRAY ELEV. READY
AND NOT   M01514	// TRAY ELEV. INITIAL HOLD
TON       T0301 50
; L18
LOAD      T0301
AND NOT   M01519	// TRAY ELEV. HOME ->
OUT       M0070A	// ONLD ELE Z POS ERR
; L19
LOAD      M0070B	// ONLD ELE Z SVD ERR
AND NOT   M00008	// RESET SW PLS
LOAD NOT  D01000.B	// TRAY ELEV. ModuleErr
AND NOT   D01000.C	// TRAY ELEV. SVD_Err
NOT
OR LOAD
AND NOT   M0070F	// ONLD ELE Z SERVO OFF
OUT       M0070B	// ONLD ELE Z SVD ERR
; L21
LOADP     T0601
LOAD      M0070C	// ONLD ELE Z NOT MV
AND NOT   M00008	// RESET SW PLS
OR LOAD
OUT       M0070C	// ONLD ELE Z NOT MV
; L23
LOAD      D01000.E	// TRAY ELEV. »óÇÑ¸®¹ÌÆ®
AND NOT   M01519	// TRAY ELEV. HOME ->
LOAD      M0070D	// ONLD ELE Z +LIMIT
AND NOT   M00008	// RESET SW PLS
OR LOAD
OUT       M0070D	// ONLD ELE Z +LIMIT
; L25
LOAD      D01000.F	// TRAY ELEV. ÇÏÇÑ¸®¹ÌÆ®
AND NOT   M01519	// TRAY ELEV. HOME ->
LOAD      M0070E	// ONLD ELE Z -LIMIT
AND NOT   M00008	// RESET SW PLS
OR LOAD
OUT       M0070E	// ONLD ELE Z -LIMIT
; L27
LOAD NOT  D01000.2	// TRAY ELEV. SVD_ON
OUT       M0070F	// ONLD ELE Z SERVO OFF

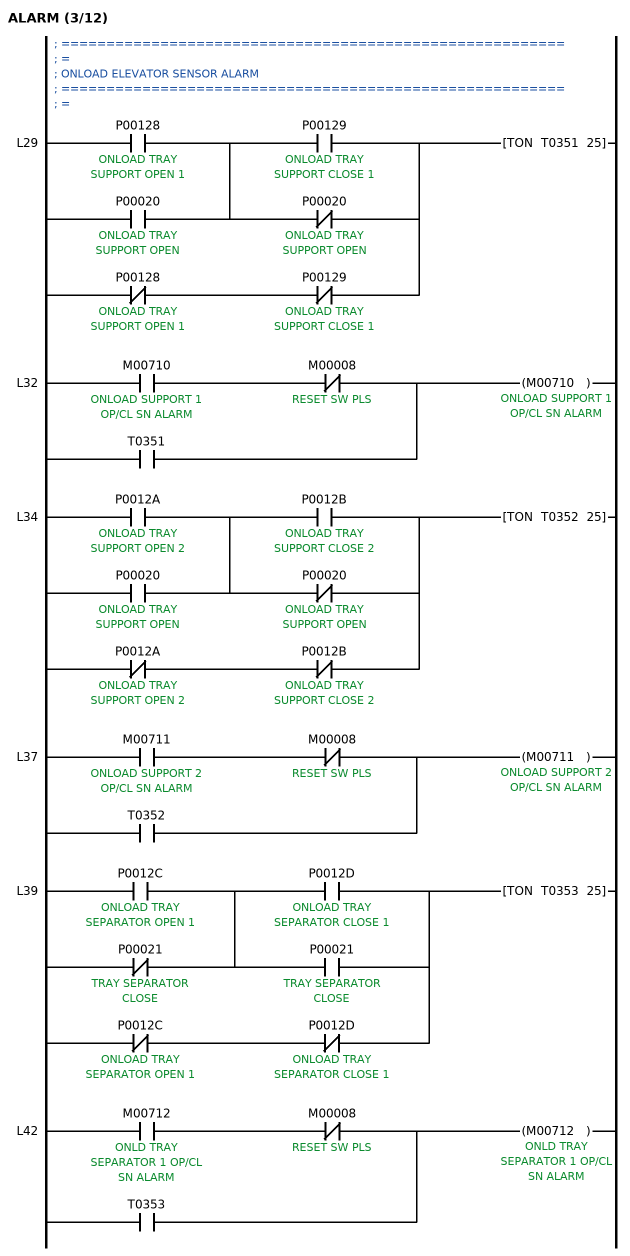
// =========================================================
// 
//        ONLOAD ELEVATOR SENSOR ALARM
// 
// =========================================================
; L29
LOAD      P00128	// ONLOAD TRAY SUPPORT OPEN 1
OR        P00020	// ONLOAD TRAY SUPPORT OPEN
LOAD      P00129	// ONLOAD TRAY SUPPORT CLOSE 1
OR NOT    P00020	// ONLOAD TRAY SUPPORT OPEN
AND LOAD
LOAD NOT  P00128	// ONLOAD TRAY SUPPORT OPEN 1
AND NOT   P00129	// ONLOAD TRAY SUPPORT CLOSE 1
OR LOAD
TON       T0351 25
; L32
LOAD      M00710	// ONLOAD SUPPORT 1 OP/CL SN ALARM
AND NOT   M00008	// RESET SW PLS
OR        T0351
OUT       M00710	// ONLOAD SUPPORT 1 OP/CL SN ALARM
; L34
LOAD      P0012A	// ONLOAD TRAY SUPPORT OPEN 2
OR        P00020	// ONLOAD TRAY SUPPORT OPEN
LOAD      P0012B	// ONLOAD TRAY SUPPORT CLOSE 2
OR NOT    P00020	// ONLOAD TRAY SUPPORT OPEN
AND LOAD
LOAD NOT  P0012A	// ONLOAD TRAY SUPPORT OPEN 2
AND NOT   P0012B	// ONLOAD TRAY SUPPORT CLOSE 2
OR LOAD
TON       T0352 25
; L37
LOAD      M00711	// ONLOAD SUPPORT 2 OP/CL SN ALARM
AND NOT   M00008	// RESET SW PLS
OR        T0352
OUT       M00711	// ONLOAD SUPPORT 2 OP/CL SN ALARM
; L39
LOAD      P0012C	// ONLOAD TRAY SEPARATOR OPEN 1
OR NOT    P00021	// TRAY SEPARATOR CLOSE
LOAD      P0012D	// ONLOAD TRAY SEPARATOR CLOSE 1
OR        P00021	// TRAY SEPARATOR CLOSE
AND LOAD
LOAD NOT  P0012C	// ONLOAD TRAY SEPARATOR OPEN 1
AND NOT   P0012D	// ONLOAD TRAY SEPARATOR CLOSE 1
OR LOAD
TON       T0353 25
; L42
LOAD      M00712	// ONLD TRAY SEPARATOR 1 OP/CL SN ALARM
AND NOT   M00008	// RESET SW PLS
OR        T0353
OUT       M00712	// ONLD TRAY SEPARATOR 1 OP/CL SN ALARM

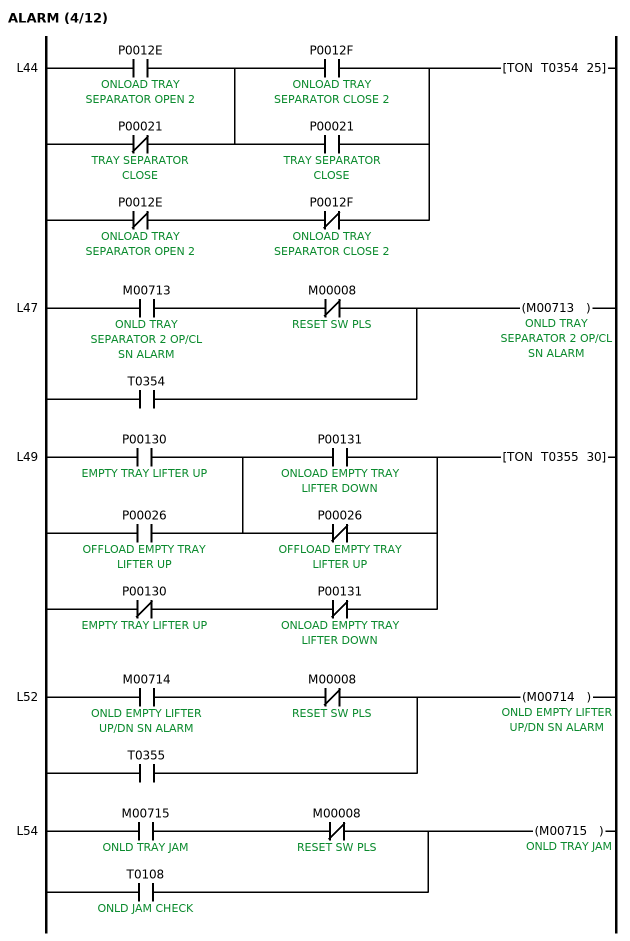
; L44
LOAD      P0012E	// ONLOAD TRAY SEPARATOR OPEN 2
OR NOT    P00021	// TRAY SEPARATOR CLOSE
LOAD      P0012F	// ONLOAD TRAY SEPARATOR CLOSE 2
OR        P00021	// TRAY SEPARATOR CLOSE
AND LOAD
LOAD NOT  P0012E	// ONLOAD TRAY SEPARATOR OPEN 2
AND NOT   P0012F	// ONLOAD TRAY SEPARATOR CLOSE 2
OR LOAD
TON       T0354 25
; L47
LOAD      M00713	// ONLD TRAY SEPARATOR 2 OP/CL SN ALARM
AND NOT   M00008	// RESET SW PLS
OR        T0354
OUT       M00713	// ONLD TRAY SEPARATOR 2 OP/CL SN ALARM
; L49
LOAD      P00130	// EMPTY TRAY LIFTER UP
OR        P00026	// OFFLOAD EMPTY TRAY LIFTER UP
LOAD      P00131	// ONLOAD EMPTY TRAY LIFTER DOWN
OR NOT    P00026	// OFFLOAD EMPTY TRAY LIFTER UP
AND LOAD
LOAD NOT  P00130	// EMPTY TRAY LIFTER UP
AND NOT   P00131	// ONLOAD EMPTY TRAY LIFTER DOWN
OR LOAD
TON       T0355 30
; L52
LOAD      M00714	// ONLD EMPTY LIFTER UP/DN SN ALARM
AND NOT   M00008	// RESET SW PLS
OR        T0355
OUT       M00714	// ONLD EMPTY LIFTER UP/DN SN ALARM
; L54
LOAD      M00715	// ONLD TRAY JAM
AND NOT   M00008	// RESET SW PLS
OR        T0108	// ONLD JAM CHECK
OUT       M00715	// ONLD TRAY JAM

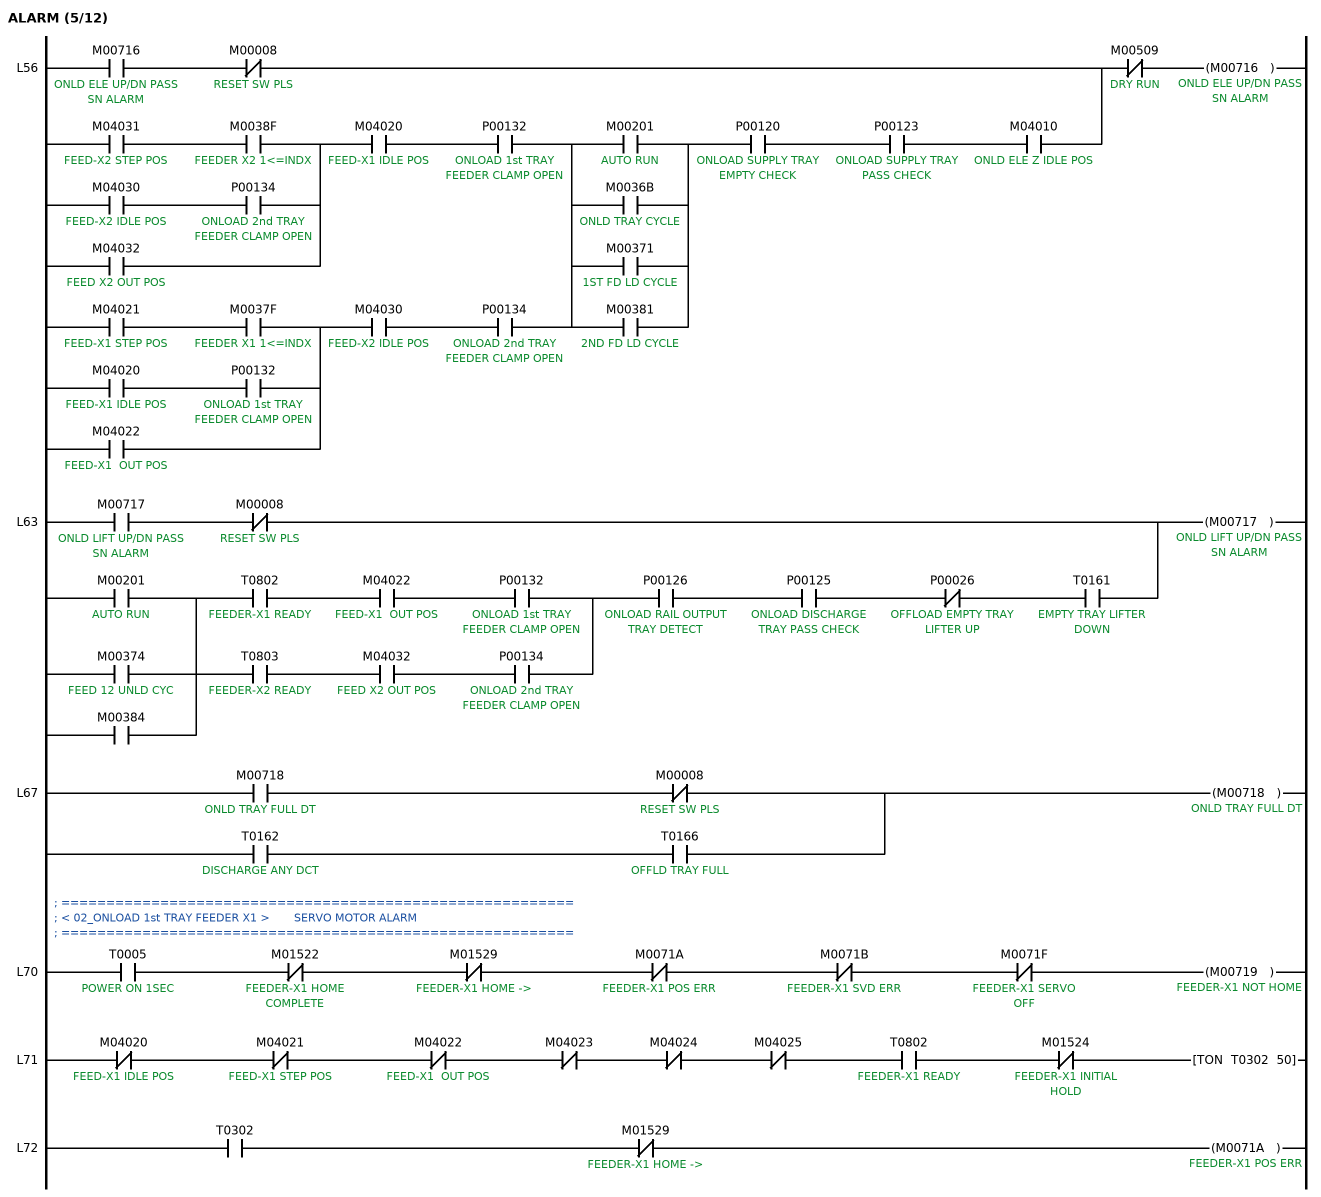
; L56
LOAD      M00716	// ONLD ELE UP/DN PASS SN ALARM
AND NOT   M00008	// RESET SW PLS
LOAD      M04031	// FEED-X2 STEP POS
AND       M0038F	// FEEDER X2 1<=INDX
LOAD      M04030	// FEED-X2 IDLE POS
AND       P00134	// ONLOAD 2nd TRAY FEEDER CLAMP OPEN
OR LOAD
OR        M04032	// FEED X2 OUT POS
AND       M04020	// FEED-X1 IDLE POS
AND       P00132	// ONLOAD 1st TRAY FEEDER CLAMP OPEN
LOAD      M04021	// FEED-X1 STEP POS
AND       M0037F	// FEEDER X1 1<=INDX
LOAD      M04020	// FEED-X1 IDLE POS
AND       P00132	// ONLOAD 1st TRAY FEEDER CLAMP OPEN
OR LOAD
OR        M04022	// FEED-X1  OUT POS
AND       M04030	// FEED-X2 IDLE POS
AND       P00134	// ONLOAD 2nd TRAY FEEDER CLAMP OPEN
OR LOAD
LOAD      M00201	// AUTO RUN
OR        M0036B	// ONLD TRAY CYCLE
OR        M00371	// 1ST FD LD CYCLE
OR        M00381	// 2ND FD LD CYCLE
AND LOAD
AND       P00120	// ONLOAD SUPPLY TRAY EMPTY CHECK
AND       P00123	// ONLOAD SUPPLY TRAY PASS CHECK
AND       M04010	// ONLD ELE Z IDLE POS
OR LOAD
AND NOT   M00509	// DRY RUN
OUT       M00716	// ONLD ELE UP/DN PASS SN ALARM
; L63
LOAD      M00717	// ONLD LIFT UP/DN PASS SN ALARM
AND NOT   M00008	// RESET SW PLS
LOAD      M00201	// AUTO RUN
OR        M00374	// FEED 12 UNLD CYC
OR        M00384
LOAD      T0802	// FEEDER-X1 READY
AND       M04022	// FEED-X1  OUT POS
AND       P00132	// ONLOAD 1st TRAY FEEDER CLAMP OPEN
LOAD      T0803	// FEEDER-X2 READY
AND       M04032	// FEED X2 OUT POS
AND       P00134	// ONLOAD 2nd TRAY FEEDER CLAMP OPEN
OR LOAD
AND LOAD
AND       P00126	// ONLOAD RAIL OUTPUT TRAY DETECT
AND       P00125	// ONLOAD DISCHARGE TRAY PASS CHECK
AND NOT   P00026	// OFFLOAD EMPTY TRAY LIFTER UP
AND       T0161	// EMPTY TRAY LIFTER DOWN
OR LOAD
OUT       M00717	// ONLD LIFT UP/DN PASS SN ALARM
; L67
LOAD      M00718	// ONLD TRAY FULL DT
AND NOT   M00008	// RESET SW PLS
LOAD      T0162	// DISCHARGE ANY DCT
AND       T0166	// OFFLD TRAY FULL
OR LOAD
OUT       M00718	// ONLD TRAY FULL DT
// =========================================================
// 
//        < 02_ONLOAD 1st TRAY FEEDER X1 >       SERVO MOTOR ALARM
// 
// =========================================================
; L70
LOAD      T0005	// POWER ON 1SEC
AND NOT   M01522	// FEEDER-X1 HOME COMPLETE
AND NOT   M01529	// FEEDER-X1 HOME ->
AND NOT   M0071A	// FEEDER-X1 POS ERR
AND NOT   M0071B	// FEEDER-X1 SVD ERR
AND NOT   M0071F	// FEEDER-X1 SERVO OFF
OUT       M00719	// FEEDER-X1 NOT HOME
; L71
LOAD NOT  M04020	// FEED-X1 IDLE POS
AND NOT   M04021	// FEED-X1 STEP POS
AND NOT   M04022	// FEED-X1  OUT POS
AND NOT   M04023
AND NOT   M04024
AND NOT   M04025
AND       T0802	// FEEDER-X1 READY
AND NOT   M01524	// FEEDER-X1 INITIAL HOLD
TON       T0302 50
; L72
LOAD      T0302
AND NOT   M01529	// FEEDER-X1 HOME ->
OUT       M0071A	// FEEDER-X1 POS ERR

